   t5[480] := -0.013076;
   t5[481] := -0.0088184;
   t5[482] := -0.0046621;
   t5[483] := -0.0006165;
   t5[484] := 0.0033093;
   t5[485] := 0.0071061;
   t5[486] := 0.0107645;
   t5[487] := 0.0142754;
   t5[488] := 0.0176295;
   t5[489] := 0.0208177;
   t5[490] := 0.023831;
   t5[491] := 0.0266696;
   t5[492] := 0.0293428;
   t5[493] := 0.0318604;
   t5[494] := 0.0342322;
   t5[495] := -0.0208986;
   t5[496] := -0.0225395;
   t5[497] := -0.0240864;
   t5[498] := -0.0255261;
   t5[499] := -0.0268454;
   t5[500] := -0.0280312;
   t5[501] := -0.0290703;
   t5[502] := -0.0299495;
   t5[503] := -0.0306555;
   t5[504] := -0.0311752;
   t5[505] := -0.0314958;
   t5[506] := -0.0316138;
   t5[507] := -0.0315351;
   t5[508] := -0.0312663;
   t5[509] := -0.0308137;
   t5[510] := -0.0136591;
   t5[511] := -0.0122989;
   t5[512] := -0.0110547;
   t5[513] := -0.0099303;
   t5[514] := -0.0089297;
   t5[515] := -0.0080568;
   t5[516] := -0.0073155;
   t5[517] := -0.0067099;
   t5[518] := -0.0062437;
   t5[519] := -0.0059209;
   t5[520] := -0.0057453;
   t5[521] := -0.0057154;
   t5[522] := -0.0058246;
   t5[523] := -0.006066;
   t5[524] := -0.0064327;
   t5[525] := -0.014299;
   t5[526] := -0.0104196;
   t5[527] := -0.0064601;
   t5[528] := -0.0024202;
   t5[529] := 0.0017005;
   t5[530] := 0.0059023;
   t5[531] := 0.0101856;
   t5[532] := 0.0145506;
   t5[533] := 0.0189979;
   t5[534] := 0.0235277;
   t5[535] := 0.0281401;
   t5[536] := 0.0328307;
   t5[537] := 0.0375902;
   t5[538] := 0.042409;
   t5[539] := 0.0472775;
   t5[540] := -0.0809446;
   t5[541] := -0.0816613;
   t5[542] := -0.0823782;
   t5[543] := -0.0831006;
   t5[544] := -0.0838339;
   t5[545] := -0.0845833;
   t5[546] := -0.0853541;
   t5[547] := -0.0861518;
   t5[548] := -0.0869815;
   t5[549] := -0.0878487;
   t5[550] := -0.0887583;
   t5[551] := -0.0897094;
   t5[552] := -0.0906944;
   t5[553] := -0.0917059;
   t5[554] := -0.092736;
   t5[555] := 0.0001257;
   t5[556] := 0.0029497;
   t5[557] := 0.0057871;
   t5[558] := 0.0086392;
   t5[559] := 0.0115078;
   t5[560] := 0.0143943;
   t5[561] := 0.0173003;
   t5[562] := 0.0202273;
   t5[563] := 0.0231768;
   t5[564] := 0.0261505;
   t5[565] := 0.0291498;
   t5[566] := 0.0321767;
   t5[567] := 0.0352333;
   t5[568] := 0.0383218;
   t5[569] := 0.0414445;
   t5[570] := -0.0673197;
   t5[571] := -0.0670321;
   t5[572] := -0.0666434;
   t5[573] := -0.0661514;
   t5[574] := -0.0655542;
   t5[575] := -0.0648497;
   t5[576] := -0.0640358;
   t5[577] := -0.0631107;
   t5[578] := -0.0620721;
   t5[579] := -0.0609182;
   t5[580] := -0.0596471;
   t5[581] := -0.0582624;
   t5[582] := -0.0567733;
   t5[583] := -0.0551894;
   t5[584] := -0.05352;
   t5[585] := 0.0792828;
   t5[586] := 0.0762561;
   t5[587] := 0.073232;
   t5[588] := 0.0702186;
   t5[589] := 0.067224;
   t5[590] := 0.0642562;
   t5[591] := 0.0613231;
   t5[592] := 0.058433;
   t5[593] := 0.0555937;
   t5[594] := 0.0528132;
   t5[595] := 0.0500996;
   t5[596] := 0.0474569;
   t5[597] := 0.0448857;
   t5[598] := 0.042386;
   t5[599] := 0.0399582;
   t5[600] := -0.1993882;
   t5[601] := -0.1970195;
   t5[602] := -0.1945705;
   t5[603] := -0.1920432;
   t5[604] := -0.1894396;
   t5[605] := -0.1867614;
   t5[606] := -0.1840106;
   t5[607] := -0.1811892;
   t5[608] := -0.1782989;
   t5[609] := -0.1753418;
   t5[610] := -0.1723197;
   t5[611] := -0.1692367;
   t5[612] := -0.1660989;
   t5[613] := -0.1629122;
   t5[614] := -0.159683;
   t5[615] := -0.110986;
   t5[616] := -0.112907;
   t5[617] := -0.1145904;
   t5[618] := -0.11603;
   t5[619] := -0.1172196;
   t5[620] := -0.118153;
   t5[621] := -0.1188239;
   t5[622] := -0.119226;
   t5[623] := -0.1193531;
   t5[624] := -0.1191991;
   t5[625] := -0.1187581;
   t5[626] := -0.1180348;
   t5[627] := -0.1170453;
   t5[628] := -0.1158056;
   t5[629] := -0.1143322;
   t5[630] := -0.0163093;
   t5[631] := -0.0198292;
   t5[632] := -0.0232166;
   t5[633] := -0.0264609;
   t5[634] := -0.0295518;
   t5[635] := -0.0324788;
   t5[636] := -0.0352314;
   t5[637] := -0.0377992;
   t5[638] := -0.0401717;
   t5[639] := -0.0423386;
   t5[640] := -0.0442896;
   t5[641] := -0.0460239;
   t5[642] := -0.0475501;
   t5[643] := -0.0488771;
   t5[644] := -0.0500139;
   t5[645] := 0.0848828;
   t5[646] := 0.0819437;
   t5[647] := 0.0790844;
   t5[648] := 0.0763136;
   t5[649] := 0.0736399;
   t5[650] := 0.0710721;
   t5[651] := 0.0686188;
   t5[652] := 0.0662886;
   t5[653] := 0.0640904;
   t5[654] := 0.0620326;
   t5[655] := 0.0601237;
   t5[656] := 0.0583629;
   t5[657] := 0.05674;
   t5[658] := 0.0552444;
   t5[659] := 0.0538658;
   t5[660] := -0.0819279;
   t5[661] := -0.0837696;
   t5[662] := -0.085415;
   t5[663] := -0.0868444;
   t5[664] := -0.088038;
   t5[665] := -0.0889764;
   t5[666] := -0.0896396;
   t5[667] := -0.0900081;
   t5[668] := -0.0900622;
   t5[669] := -0.0897822;
   t5[670] := -0.0891493;
   t5[671] := -0.0881638;
   t5[672] := -0.0868462;
   t5[673] := -0.0852177;
   t5[674] := -0.0832996;
   t5[675] := -0.0222091;
   t5[676] := -0.019204;
   t5[677] := -0.0163363;
   t5[678] := -0.0136269;
   t5[679] := -0.0110964;
   t5[680] := -0.0087656;
   t5[681] := -0.0066552;
   t5[682] := -0.004786;
   t5[683] := -0.0031786;
   t5[684] := -0.0018538;
   t5[685] := -0.0008317;
   t5[686] := -0.0001178;
   t5[687] := 0.0002977;
   t5[688] := 0.0004254;
   t5[689] := 0.0002755;
   t5[690] := -0.0469918;
   t5[691] := -0.0436484;
   t5[692] := -0.0405246;
   t5[693] := -0.0376308;
   t5[694] := -0.0349775;
   t5[695] := -0.0325752;
   t5[696] := -0.0304344;
   t5[697] := -0.0285657;
   t5[698] := -0.0269795;
   t5[699] := -0.0256863;
   t5[700] := -0.0246962;
   t5[701] := -0.0240066;
   t5[702] := -0.0236022;
   t5[703] := -0.0234672;
   t5[704] := -0.0235855;
   t5[705] := 0.0315658;
   t5[706] := 0.0328791;
   t5[707] := 0.0340612;
   t5[708] := 0.0351116;
   t5[709] := 0.0360298;
   t5[710] := 0.0368152;
   t5[711] := 0.0374672;
   t5[712] := 0.0379854;
   t5[713] := 0.0383692;
   t5[714] := 0.038618;
   t5[715] := 0.0387315;
   t5[716] := 0.0387144;
   t5[717] := 0.0385764;
   t5[718] := 0.0383273;
   t5[719] := 0.0379772;
   t5[720] := 0.0589575;
   t5[721] := 0.0571638;
   t5[722] := 0.0552337;
   t5[723] := 0.0531697;
   t5[724] := 0.0509741;
   t5[725] := 0.0486495;
   t5[726] := 0.0461984;
   t5[727] := 0.0436231;
   t5[728] := 0.0409261;
   t5[729] := 0.03811;
   t5[730] := 0.0351772;
   t5[731] := 0.0321336;
   t5[732] := 0.0289883;
   t5[733] := 0.0257505;
   t5[734] := 0.0224294;
   t5[735] := -0.0370074;
   t5[736] := -0.0344528;
   t5[737] := -0.0317711;
   t5[738] := -0.0289586;
   t5[739] := -0.0260112;
   t5[740] := -0.022925;
   t5[741] := -0.0196963;
   t5[742] := -0.016321;
   t5[743] := -0.0127952;
   t5[744] := -0.0091151;
   t5[745] := -0.005277;
   t5[746] := -0.0012858;
   t5[747] := 0.0028455;
   t5[748] := 0.007103;
   t5[749] := 0.0114734;
   t5[750] := -0.0503424;
   t5[751] := -0.0554995;
   t5[752] := -0.0605443;
   t5[753] := -0.0654624;
   t5[754] := -0.0702395;
   t5[755] := -0.0748614;
   t5[756] := -0.0793139;
   t5[757] := -0.0835825;
   t5[758] := -0.087653;
   t5[759] := -0.0915111;
   t5[760] := -0.095143;
   t5[761] := -0.0985424;
   t5[762] := -0.1017114;
   t5[763] := -0.1046524;
   t5[764] := -0.1073677;
   t5[765] := -0.1648159;
   t5[766] := -0.1596806;
   t5[767] := -0.1543417;
   t5[768] := -0.1488126;
   t5[769] := -0.1431066;
   t5[770] := -0.1372371;
   t5[771] := -0.1312175;
   t5[772] := -0.1250611;
   t5[773] := -0.1187812;
   t5[774] := -0.1123913;
   t5[775] := -0.1059046;
   t5[776] := -0.0993333;
   t5[777] := -0.0926887;
   t5[778] := -0.0859816;
   t5[779] := -0.0792232;
   t5[780] := -0.0904827;
   t5[781] := -0.0898896;
   t5[782] := -0.0893127;
   t5[783] := -0.0887551;
   t5[784] := -0.0882202;
   t5[785] := -0.0877112;
   t5[786] := -0.0872314;
   t5[787] := -0.0867841;
   t5[788] := -0.0863725;
   t5[789] := -0.0859999;
   t5[790] := -0.0856695;
   t5[791] := -0.0853802;
   t5[792] := -0.0851272;
   t5[793] := -0.0849053;
   t5[794] := -0.0847093;
   t5[795] := -0.0673839;
   t5[796] := -0.0627446;
   t5[797] := -0.0580462;
   t5[798] := -0.0533;
   t5[799] := -0.0485171;
   t5[800] := -0.0437086;
   t5[801] := -0.0388857;
   t5[802] := -0.0340594;
   t5[803] := -0.0292411;
   t5[804] := -0.0244417;
   t5[805] := -0.0196723;
   t5[806] := -0.0149416;
   t5[807] := -0.0102555;
   t5[808] := -0.0056201;
   t5[809] := -0.0010412;
   t5[810] := 0.075334;
   t5[811] := 0.0749833;
   t5[812] := 0.0743661;
   t5[813] := 0.0734706;
   t5[814] := 0.072285;
   t5[815] := 0.0707974;
   t5[816] := 0.068996;
   t5[817] := 0.0668689;
   t5[818] := 0.0644045;
   t5[819] := 0.0615908;
   t5[820] := 0.0584166;
   t5[821] := 0.0548866;
   t5[822] := 0.0510212;
   t5[823] := 0.0468419;
   t5[824] := 0.04237;
   t5[825] := -0.1063465;
   t5[826] := -0.1045535;
   t5[827] := -0.1026798;
   t5[828] := -0.1007291;
   t5[829] := -0.0987055;
   t5[830] := -0.0966127;
   t5[831] := -0.0944546;
   t5[832] := -0.092235;
   t5[833] := -0.0899577;
   t5[834] := -0.0876267;
   t5[835] := -0.0852457;
   t5[836] := -0.0828167;
   t5[837] := -0.0803401;
   t5[838] := -0.077816;
   t5[839] := -0.0752449;
   t5[840] := 0.0025241;
   t5[841] := 0.0003729;
   t5[842] := -0.0018117;
   t5[843] := -0.0040243;
   t5[844] := -0.0062591;
   t5[845] := -0.0085107;
   t5[846] := -0.0107734;
   t5[847] := -0.0130416;
   t5[848] := -0.0153097;
   t5[849] := -0.0175722;
   t5[850] := -0.0198235;
   t5[851] := -0.0220606;
   t5[852] := -0.0242824;
   t5[853] := -0.0264882;
   t5[854] := -0.0286772;
   t5[855] := -0.0587365;
   t5[856] := -0.0658987;
   t5[857] := -0.0729648;
   t5[858] := -0.07991;
   t5[859] := -0.0867094;
   t5[860] := -0.0933378;
   t5[861] := -0.0997704;
   t5[862] := -0.1059823;
   t5[863] := -0.1119484;
   t5[864] := -0.1176438;
   t5[865] := -0.1230443;
   t5[866] := -0.1281403;
   t5[867] := -0.1329374;
   t5[868] := -0.137442;
   t5[869] := -0.1416606;
   t5[870] := -0.0241061;
   t5[871] := -0.0227329;
   t5[872] := -0.0212774;
   t5[873] := -0.0197337;
   t5[874] := -0.0180954;
   t5[875] := -0.0163565;
   t5[876] := -0.0145109;
   t5[877] := -0.0125525;
   t5[878] := -0.0104751;
   t5[879] := -0.0082726;
   t5[880] := -0.0059392;
   t5[881] := -0.0034767;
   t5[882] := -0.0008946;
   t5[883] := 0.001797;
   t5[884] := 0.0045883;
   t5[885] := -0.016338;
   t5[886] := -0.0135221;
   t5[887] := -0.0107115;
   t5[888] := -0.0079037;
   t5[889] := -0.0050963;
   t5[890] := -0.0022869;
   t5[891] := 0.0005271;
   t5[892] := 0.0033482;
   t5[893] := 0.0061787;
   t5[894] := 0.0090212;
   t5[895] := 0.011878;
   t5[896] := 0.0147486;
   t5[897] := 0.0176293;
   t5[898] := 0.0205164;
   t5[899] := 0.0234063;
   t5[900] := -0.0519279;
   t5[901] := -0.056473;
   t5[902] := -0.0609004;
   t5[903] := -0.0652012;
   t5[904] := -0.0693667;
   t5[905] := -0.0733882;
   t5[906] := -0.0772569;
   t5[907] := -0.0809641;
   t5[908] := -0.0845011;
   t5[909] := -0.087859;
   t5[910] := -0.0910294;
   t5[911] := -0.0940104;
   t5[912] := -0.0968068;
   t5[913] := -0.0994238;
   t5[914] := -0.1018665;
   t5[915] := 0.142846;
   t5[916] := 0.1405271;
   t5[917] := 0.1380653;
   t5[918] := 0.1354591;
   t5[919] := 0.1327065;
   t5[920] := 0.129806;
   t5[921] := 0.1267559;
   t5[922] := 0.1235543;
   t5[923] := 0.1201996;
   t5[924] := 0.11669;
   t5[925] := 0.1130242;
   t5[926] := 0.109206;
   t5[927] := 0.1052453;
   t5[928] := 0.1011521;
   t5[929] := 0.0969364;
   t5[930] := -0.0299947;
   t5[931] := -0.0294521;
   t5[932] := -0.0288785;
   t5[933] := -0.0282723;
   t5[934] := -0.0276319;
   t5[935] := -0.0269553;
   t5[936] := -0.0262411;
   t5[937] := -0.0254874;
   t5[938] := -0.0246926;
   t5[939] := -0.0238549;
   t5[940] := -0.0229728;
   t5[941] := -0.0220476;
   t5[942] := -0.0210837;
   t5[943] := -0.0200855;
   t5[944] := -0.0190576;
   t5[945] := -0.0100999;
   t5[946] := -0.0030712;
   t5[947] := 0.0037406;
   t5[948] := 0.0103103;
   t5[949] := 0.0166126;
   t5[950] := 0.0226221;
   t5[951] := 0.0283136;
   t5[952] := 0.0336617;
   t5[953] := 0.038641;
   t5[954] := 0.0432264;
   t5[955] := 0.0473932;
   t5[956] := 0.0511381;
   t5[957] := 0.054479;
   t5[958] := 0.0574348;
   t5[959] := 0.0600244;
   w6[0] := 0.0254122;
   w6[1] := -0.4251655;
   w6[2] := -0.4513899;
   w6[3] := 0.0262705;
   w6[4] := 0.3702881;
   w6[5] := -0.1208161;
   w6[6] := -0.2231239;
   w6[7] := 0.2512441;
   w6[8] := -0.3278799;
   w6[9] := 0.2889541;
   w6[10] := -0.0654242;
   w6[11] := 0.1067281;
   w6[12] := 0.2623815;
   w6[13] := -0.1798091;
   w6[14] := -0.3070911;
   w6[15] := -0.4204447;
   w6[16] := 0.5762351;
   w6[17] := -1.090657;
   w6[18] := -0.2690518;
   w6[19] := -0.6730261;
   w6[20] := -0.0514923;
   w6[21] := -0.4457789;
   w6[22] := 0.5072183;
   w6[23] := -0.0549661;
   w6[24] := 0.3812394;
   w6[25] := -0.606307;
   w6[26] := 0.1917919;
   w6[27] := 0.1525442;
   w6[28] := -0.4219312;
   w6[29] := 0.338313;
   w6[30] := 0.1919874;
   w6[31] := -0.3457294;
   w6[32] := 0.1728978;
   w6[33] := 0.5825878;
   w6[34] := 0.7331663;
   w6[35] := 0.4268312;
   w6[36] := -0.0077422;
   w6[37] := 0.4766487;
   w6[38] := 0.102607;
   w6[39] := -0.5723706;
   w6[40] := 0.0728498;
   w6[41] := 0.4253429;
   w6[42] := -0.3637053;
   w6[43] := -0.6206156;
   w6[44] := 0.2656944;
   w6[45] := -0.3130539;
   w6[46] := 0.2033212;
   w6[47] := 0.1327122;
   w6[48] := -0.709101;
   w6[49] := 0.7231103;
   w6[50] := -0.2214241;
   w6[51] := 0.4491622;
   w6[52] := -0.3655713;
   w6[53] := 0.4263724;
   w6[54] := 0.0266531;
   w6[55] := 0.4637966;
   w6[56] := -0.3418979;
   w6[57] := -0.2391363;
   w6[58] := 0.4152579;
   w6[59] := 0.2146362;
   w6[60] := -0.3901598;
   w6[61] := -0.1938754;
   w6[62] := -0.561949;
   w6[63] := 0.4047181;
END_DATA_BLOCK

DATA_BLOCK "NeuroPLC_MLP_Weights"   // DB3
{ S7_Optimized_Access := 'FALSE' }
VERSION : 0.1
   VAR
      w0 : Array[0..895] of Real;   // W(32x28)
      b1 : Array[0..31] of Real;   // bias(32)
      w2 : Array[0..511] of Real;   // W(16x32)
      b3 : Array[0..15] of Real;   // bias(16)
      w4 : Array[0..63] of Real;   // W(4x16)
      b5 : Array[0..3] of Real;   // bias(4)
   END_VAR
BEGIN
   w0[0] := 0.5694862;
   w0[1] := -0.0095692;
   w0[2] := 0.7619486;
   w0[3] := 0.2215109;
   w0[4] := -0.3561512;
   w0[5] := -0.2522623;
   w0[6] := 0.2582799;
   w0[7] := 0.0099258;
   w0[8] := 0.3836571;
   w0[9] := -0.0658457;
   w0[10] := 0.1010401;
   w0[11] := -0.2984352;
   w0[12] := 0.1934527;
   w0[13] := -0.264014;
   w0[14] := 0.1362384;
   w0[15] := -0.0190728;
   w0[16] := -0.2375232;
   w0[17] := -0.1084833;
   w0[18] := -0.3846658;
   w0[19] := 0.3771667;
   w0[20] := -0.1136759;
   w0[21] := -0.1259104;
   w0[22] := -0.1682155;
   w0[23] := 0.4097499;
   w0[24] := -0.2194012;
   w0[25] := -0.2356472;
   w0[26] := -0.1771912;
   w0[27] := 0.1675407;
   w0[28] := 0.1454716;
   w0[29] := -0.3696787;
   w0[30] := -0.2783369;
   w0[31] := -0.1873165;
   w0[32] := 0.0781848;
   w0[33] := -0.3527579;
   w0[34] := -0.2131715;
   w0[35] := -0.413968;
   w0[36] := -0.5927966;
   w0[37] := 0.3198802;
   w0[38] := -0.5640871;
   w0[39] := -0.2003005;
   w0[40] := 0.1832723;
   w0[41] := 0.2237836;
   w0[42] := 0.1929916;
   w0[43] := 0.2185234;
   w0[44] := 0.1214973;
   w0[45] := 0.0208249;
   w0[46] := 0.2776418;
   w0[47] := 0.6831574;
   w0[48] := -0.1655439;
   w0[49] := -0.2658227;
   w0[50] := -0.2709237;
   w0[51] := 0.098671;
   w0[52] := 0.1128972;
   w0[53] := -0.2047481;
   w0[54] := -0.3872808;
   w0[55] := 0.1596099;
   w0[56] := -0.2523361;
   w0[57] := 0.2758174;
   w0[58] := 0.2686562;
   w0[59] := -0.5177624;
   w0[60] := -0.1129441;
   w0[61] := -0.21921;
   w0[62] := 0.3343761;
   w0[63] := -0.0422801;
   w0[64] := -0.3068857;
   w0[65] := 0.2210509;
   w0[66] := -0.5496964;
   w0[67] := 0.3709493;
   w0[68] := 0.0747587;
   w0[69] := -0.1170707;
   w0[70] := -0.319511;
   w0[71] := 0.0277475;
   w0[72] := -0.2577946;
   w0[73] := 0.0641775;
   w0[74] := 0.2055912;
   w0[75] := 0.6039576;
   w0[76] := -0.5010191;
   w0[77] := 0.0377836;
   w0[78] := 0.2038942;
   w0[79] := -0.0376425;
   w0[80] := 0.1546009;
   w0[81] := 0.3260912;
   w0[82] := -0.1506072;
   w0[83] := 0.0569262;
   w0[84] := -0.1928782;
   w0[85] := -0.198454;
   w0[86] := -0.0539345;
   w0[87] := 0.3094364;
   w0[88] := 0.2289592;
   w0[89] := -0.425005;
   w0[90] := -0.0399776;
   w0[91] := 0.0658291;
   w0[92] := 0.2534966;
   w0[93] := -0.0973715;
   w0[94] := -0.3647969;
   w0[95] := -0.015606;
   w0[96] := -0.5209337;
   w0[97] := 0.2564455;
   w0[98] := 0.1338747;
   w0[99] := 0.3502659;
   w0[100] := -0.3756513;
   w0[101] := 0.253089;
   w0[102] := 0.0984663;
   w0[103] := 0.6602526;
   w0[104] := 0.3365156;
   w0[105] := -0.2521311;
   w0[106] := 0.0946512;
   w0[107] := -0.6085349;
   w0[108] := -0.5372492;
   w0[109] := 0.0455726;
   w0[110] := -0.0786947;
   w0[111] := 0.0370381;
   w0[112] := -0.585835;
   w0[113] := -0.7779619;
   w0[114] := -0.7385424;
   w0[115] := -0.207106;
   w0[116] := 0.2831336;
   w0[117] := 0.3243212;
   w0[118] := 0.2366221;
   w0[119] := -0.2105746;
   w0[120] := -0.3834608;
   w0[121] := -0.6828474;
   w0[122] := 0.1007835;
   w0[123] := 0.0381121;
   w0[124] := 0.3126857;
   w0[125] := 0.0975034;
   w0[126] := 0.0499541;
   w0[127] := -0.0530838;
   w0[128] := 0.0799674;
   w0[129] := -0.1505451;
   w0[130] := -0.4892448;
   w0[131] := -0.3954702;
   w0[132] := 0.1594549;
   w0[133] := 0.2307071;
   w0[134] := -0.0041823;
   w0[135] := 0.5944483;
   w0[136] := -0.2759206;
   w0[137] := -0.4257804;
   w0[138] := -0.3279784;
   w0[139] := -0.297798;
   w0[140] := 0.0038754;
   w0[141] := 0.3761657;
   w0[142] := 0.4177073;
   w0[143] := 0.0741864;
   w0[144] := 0.3750937;
   w0[145] := 0.2039272;
   w0[146] := -0.2429399;
   w0[147] := -0.3849822;
   w0[148] := 0.1600508;
   w0[149] := -0.1581226;
   w0[150] := -0.0233814;
   w0[151] := -0.1151747;
   w0[152] := -0.5731639;
   w0[153] := -0.0274457;
   w0[154] := 0.1195597;
   w0[155] := -0.2395748;
   w0[156] := 0.2293357;
   w0[157] := -0.0251415;
   w0[158] := 0.3937997;
   w0[159] := -0.1454628;
   w0[160] := -0.0673693;
   w0[161] := 0.2948158;
   w0[162] := 0.5630679;
   w0[163] := -0.3092144;
   w0[164] := 0.1832785;
   w0[165] := 0.004312;
   w0[166] := 0.0011036;
   w0[167] := 0.2549984;
   w0[168] := 0.1242365;
   w0[169] := -0.1573328;
   w0[170] := 0.1472307;
   w0[171] := 0.2971004;
   w0[172] := 0.1052006;
   w0[173] := 0.3616425;
   w0[174] := -0.1347494;
   w0[175] := -0.3794992;
   w0[176] := 0.5467421;
   w0[177] := -0.1476457;
   w0[178] := 0.3496484;
   w0[179] := -0.0583753;
   w0[180] := 0.2853532;
   w0[181] := -0.3058073;
   w0[182] := -0.1615329;
   w0[183] := -0.522915;
   w0[184] := 0.2140338;
   w0[185] := -0.2294949;
   w0[186] := 0.2921923;
   w0[187] := 0.0373898;
   w0[188] := 0.3493846;
   w0[189] := 0.5938788;
   w0[190] := 0.0955027;
   w0[191] := -0.1719695;
   w0[192] := 0.6582399;
   w0[193] := -0.491165;
   w0[194] := 0.126987;
   w0[195] := -0.412937;
   w0[196] := -0.273549;
   w0[197] := -0.215566;
   w0[198] := 0.4269275;
   w0[199] := -0.1273027;
   w0[200] := -0.2414422;
   w0[201] := -0.3611139;
   w0[202] := 0.6480063;
   w0[203] := 0.3808921;
   w0[204] := -0.2189153;
   w0[205] := 0.0094489;
   w0[206] := 0.6784652;
   w0[207] := 0.3757944;
   w0[208] := 0.5965886;
   w0[209] := 0.3704935;
   w0[210] := 0.3205929;
   w0[211] := 0.2190031;
   w0[212] := -0.3913886;
   w0[213] := 0.2046225;
   w0[214] := 0.7660633;
   w0[215] := 0.5648795;
   w0[216] := 0.0447379;
   w0[217] := -0.1363681;
   w0[218] := -0.1653181;
   w0[219] := -0.3211187;
   w0[220] := 0.0557173;
   w0[221] := -0.677563;
   w0[222] := 0.2077208;
   w0[223] := 0.1863764;
   w0[224] := 0.0122372;
   w0[225] := -0.1510706;
   w0[226] := -0.0393031;
   w0[227] := -0.237385;
   w0[228] := 0.3297745;
   w0[229] := -0.3327326;
   w0[230] := -0.1183226;
   w0[231] := 0.3871697;
   w0[232] := -0.448105;
   w0[233] := -0.2065133;
   w0[234] := 0.1012533;
   w0[235] := -0.2578072;
   w0[236] := 0.0634624;
   w0[237] := -0.1246978;
   w0[238] := 0.1465549;
   w0[239] := -0.5023389;
   w0[240] := 0.0640146;
   w0[241] := 0.1963426;
   w0[242] := 0.6648222;
   w0[243] := -0.6102669;
   w0[244] := -0.28719;
   w0[245] := -0.3684005;
   w0[246] := -0.4533643;
   w0[247] := -0.1819637;
   w0[248] := -0.3802012;
   w0[249] := 0.4682154;
   w0[250] := 0.1991423;
   w0[251] := 0.5698866;
   w0[252] := 0.3063245;
   w0[253] := 0.1672625;
   w0[254] := 0.261124;
   w0[255] := -0.6845852;
   w0[256] := -0.1005014;
   w0[257] := -0.6641653;
   w0[258] := -0.254451;
   w0[259] := 0.1954752;
   w0[260] := -0.2994281;
   w0[261] := 0.3571715;
   w0[262] := -0.0372742;
   w0[263] := -0.0310561;
   w0[264] := 0.1959654;
   w0[265] := -0.1060541;
   w0[266] := 0.3827632;
   w0[267] := -0.3923316;
   w0[268] := -0.592409;
   w0[269] := 0.0670658;
   w0[270] := 0.3532278;
   w0[271] := 0.6439264;
   w0[272] := 0.1193878;
   w0[273] := -0.5490641;
   w0[274] := -0.6517076;
   w0[275] := 0.2266813;
   w0[276] := 0.273508;
   w0[277] := 0.2562127;
   w0[278] := 0.3711089;
   w0[279] := -0.0201157;
   w0[280] := 0.5907255;
   w0[281] := 0.3026478;
   w0[282] := 0.087949;
   w0[283] := -0.1103418;
   w0[284] := 0.0830003;
   w0[285] := 0.0901832;
   w0[286] := 0.4872787;
   w0[287] := -0.4248994;
   w0[288] := 0.6916616;
   w0[289] := 0.0068263;
   w0[290] := 0.0377772;
   w0[291] := -0.345046;
   w0[292] := 0.5848706;
   w0[293] := -0.0756037;
   w0[294] := 0.0390328;
   w0[295] := -0.4139087;
   w0[296] := -0.1527735;
   w0[297] := -0.2285863;
   w0[298] := 0.3310088;
   w0[299] := 0.2031009;
   w0[300] := -0.5309294;
   w0[301] := -0.4607368;
   w0[302] := 0.1824918;
   w0[303] := -0.1911459;
   w0[304] := -0.1732452;
   w0[305] := -0.3283744;
   w0[306] := -0.0425148;
   w0[307] := -0.075475;
   w0[308] := -0.075183;
   w0[309] := -0.0057766;
   w0[310] := -0.0669558;
   w0[311] := -0.0518108;
   w0[312] := -0.1100485;
   w0[313] := 0.4202482;
   w0[314] := 0.1722786;
   w0[315] := 0.254064;
   w0[316] := -0.2125306;
   w0[317] := -0.3108644;
   w0[318] := -0.1653187;
   w0[319] := 0.0082027;
   w0[320] := 0.1613134;
   w0[321] := 0.5696448;
   w0[322] := 0.4734836;
   w0[323] := -0.1820288;
   w0[324] := -0.0202256;
   w0[325] := 0.2319008;
   w0[326] := 0.6178575;
   w0[327] := -0.1729726;
   w0[328] := -0.5705087;
   w0[329] := -0.4175466;
   w0[330] := -0.0846097;
   w0[331] := -0.4305633;
   w0[332] := -0.0297265;
   w0[333] := -0.2146564;
   w0[334] := -0.0228577;
   w0[335] := 0.4386194;
   w0[336] := 0.1366172;
   w0[337] := 0.1275948;
   w0[338] := 0.2872518;
   w0[339] := -0.046949;
   w0[340] := -0.3430789;
   w0[341] := -0.2333279;
   w0[342] := -0.0942715;
   w0[343] := -0.6695372;
   w0[344] := 0.3036573;
   w0[345] := 0.6706407;
   w0[346] := 0.4867018;
   w0[347] := 0.2229243;
   w0[348] := 0.1479198;
   w0[349] := 0.4786703;
   w0[350] := -0.1235309;
   w0[351] := -0.1444162;
   w0[352] := -0.1594525;
   w0[353] := 0.0118241;
   w0[354] := 0.3302614;
   w0[355] := 0.4612524;
   w0[356] := -0.1728074;
   w0[357] := -0.4940682;
   w0[358] := 0.266313;
   w0[359] := 0.4213447;
   w0[360] := 0.155972;
   w0[361] := 0.0927116;
   w0[362] := 0.2581408;
   w0[363] := 0.1484697;
   w0[364] := 0.5596921;
   w0[365] := 0.6450443;
   w0[366] := 0.2316463;
   w0[367] := -0.3064318;
   w0[368] := 0.315403;
   w0[369] := 0.2504337;
   w0[370] := 0.2270162;
   w0[371] := -0.2362736;
   w0[372] := -0.1822204;
   w0[373] := 0.7585521;
   w0[374] := 0.2454521;
   w0[375] := -0.3572387;
   w0[376] := 0.1800293;
   w0[377] := 0.1965537;
   w0[378] := 0.1946464;
   w0[379] := 0.1738928;
   w0[380] := -0.1159788;
   w0[381] := -0.1791228;
   w0[382] := 0.3109314;
   w0[383] := 0.1039406;
   w0[384] := -0.255849;
   w0[385] := -0.4132357;
   w0[386] := -0.1826324;
   w0[387] := -0.0949509;
   w0[388] := 0.075463;
   w0[389] := -0.4951166;
   w0[390] := -0.0366096;
   w0[391] := -0.5241205;
   w0[392] := 0.0701182;
   w0[393] := 0.5458165;
   w0[394] := -0.3082272;
   w0[395] := -0.162029;
   w0[396] := 0.2685293;
   w0[397] := -0.1115321;
   w0[398] := 0.5528188;
   w0[399] := 0.1818966;
   w0[400] := -0.270587;
   w0[401] := -0.4477837;
   w0[402] := -0.3260813;
   w0[403] := -0.1751753;
   w0[404] := 0.3439055;
   w0[405] := 0.369066;
   w0[406] := -0.0775537;
   w0[407] := -0.3291571;
   w0[408] := 0.396657;
   w0[409] := 0.3747428;
   w0[410] := 0.2037812;
   w0[411] := 0.506327;
   w0[412] := -0.0363616;
   w0[413] := -0.0945516;
   w0[414] := -0.2667596;
   w0[415] := -0.1880456;
   w0[416] := 0.2148547;
   w0[417] := -0.659289;
   w0[418] := -0.2238534;
   w0[419] := -0.2862469;
   w0[420] := -0.8308039;
   w0[421] := -0.4430834;
   w0[422] := -0.0302747;
   w0[423] := 0.091846;
   w0[424] := -0.3334551;
   w0[425] := -0.1804388;
   w0[426] := -0.1097601;
   w0[427] := 0.3427432;
   w0[428] := 0.0736062;
   w0[429] := -0.6790179;
   w0[430] := -0.243052;
   w0[431] := -0.2084594;
   w0[432] := 0.1491454;
   w0[433] := -0.0083196;
   w0[434] := 0.2553293;
   w0[435] := 0.1678275;
   w0[436] := 0.0936099;
   w0[437] := 0.1736043;
   w0[438] := -0.5376837;
   w0[439] := -0.4510113;
   w0[440] := -0.3174161;
   w0[441] := 0.2371299;
   w0[442] := 0.3883051;
   w0[443] := 0.3464468;
   w0[444] := 0.1098732;
   w0[445] := 0.0205052;
   w0[446] := -0.2641115;
   w0[447] := -0.3012585;
   w0[448] := -0.5463231;
   w0[449] := -0.0684724;
   w0[450] := -0.1422806;
   w0[451] := -0.2644515;
   w0[452] := -0.4767578;
   w0[453] := -0.4182616;
   w0[454] := -0.4673964;
   w0[455] := -0.0129319;
   w0[456] := -0.5374129;
   w0[457] := -0.1050398;
   w0[458] := 0.0632549;
   w0[459] := 0.0568505;
   w0[460] := 0.2111508;
   w0[461] := 0.3917949;
   w0[462] := -0.0330271;
   w0[463] := 0.2814879;
   w0[464] := -0.3214771;
   w0[465] := 0.343051;
   w0[466] := -0.3870021;
   w0[467] := -0.4042188;
   w0[468] := 0.1747253;
   w0[469] := 0.3262924;
   w0[470] := 0.5594077;
   w0[471] := 0.0277393;
   w0[472] := -0.2604083;
   w0[473] := 0.0503597;
   w0[474] := 0.3725081;
   w0[475] := -0.0544451;
   w0[476] := 0.0951887;
   w0[477] := -0.5271522;
   w0[478] := -0.3720489;
   w0[479] := 0.0333015;
   w0[480] := 0.3407656;
   w0[481] := -0.0524092;
   w0[482] := -0.394772;
   w0[483] := 0.0632993;
   w0[484] := -0.4918242;
   w0[485] := -0.0408889;
   w0[486] := 0.5603451;
   w0[487] := 0.3429145;
   w0[488] := -0.0672607;
   w0[489] := -0.3218429;
   w0[490] := -0.3621323;
   w0[491] := -0.5524946;
   w0[492] := 0.3105496;
   w0[493] := 0.3352183;
   w0[494] := -0.6259544;
   w0[495] := -0.1107638;
   w0[496] := 0.0901521;
   w0[497] := 0.00385;
   w0[498] := 0.5420415;
   w0[499] := 0.2380718;
   w0[500] := -0.0511688;
   w0[501] := -0.077146;
   w0[502] := -0.0791493;
   w0[503] := -0.1069665;
   w0[504] := 0.6399192;
   w0[505] := -0.0014034;
   w0[506] := 0.3290343;
   w0[507] := -0.3565734;
   w0[508] := 0.2305476;
   w0[509] := -0.0417552;
   w0[510] := 0.294279;
   w0[511] := -0.1355964;
   w0[512] := 0.0557771;
   w0[513] := 0.3271682;
   w0[514] := -0.3025698;
   w0[515] := 0.28975;
   w0[516] := 0.1278277;
   w0[517] := -0.1560617;
   w0[518] := 0.2582703;
   w0[519] := -0.0549245;
   w0[520] := -0.0921321;
   w0[521] := 0.4996554;
   w0[522] := 0.0836308;
   w0[523] := 0.2032579;
   w0[524] := -0.1741465;
   w0[525] := -0.2436171;
   w0[526] := -0.3661414;
   w0[527] := -0.2924559;
   w0[528] := -0.4407195;
   w0[529] := 0.2304931;
   w0[530] := -0.2509898;
   w0[531] := -0.688146;
   w0[532] := 0.1500384;
   w0[533] := 0.4429501;
   w0[534] := 0.5444623;
   w0[535] := 0.0644146;
   w0[536] := 0.1564979;
   w0[537] := 0.1936211;
   w0[538] := -0.2217757;
   w0[539] := 0.163296;
   w0[540] := 0.0949209;
   w0[541] := 0.5449093;
   w0[542] := 0.3260632;
   w0[543] := 0.4177442;
   w0[544] := -0.1678705;
   w0[545] := -0.4614883;
   w0[546] := -0.1780888;
   w0[547] := 0.0282706;
   w0[548] := -0.3548764;
   w0[549] := 0.1119965;
   w0[550] := -0.6278588;
   w0[551] := -0.2857478;
   w0[552] := 0.3291071;
   w0[553] := -0.2958602;
   w0[554] := -0.2171935;
   w0[555] := 0.0488607;
   w0[556] := -0.2721503;
   w0[557] := -0.0109805;
   w0[558] := -0.2872001;
   w0[559] := -0.3800366;
   w0[560] := 0.7377275;
   w0[561] := 0.5175216;
   w0[562] := 0.4534726;
   w0[563] := 0.2131705;
   w0[564] := 0.1694544;
   w0[565] := 0.1088488;
   w0[566] := 0.2956495;
   w0[567] := -0.1219863;
   w0[568] := 0.4281839;
   w0[569] := 0.0482728;
   w0[570] := 0.326145;
   w0[571] := 0.0147065;
   w0[572] := 0.0197347;
   w0[573] := -0.2837075;
   w0[574] := -0.2223815;
   w0[575] := -0.3011971;
   w0[576] := 0.4010099;
   w0[577] := 0.3606303;
   w0[578] := 0.5675586;
   w0[579] := -0.1933776;
   w0[580] := 0.1411208;
   w0[581] := 0.4412328;
   w0[582] := -0.3157989;
   w0[583] := 0.0737199;
   w0[584] := 0.2547267;
   w0[585] := -0.4104514;
   w0[586] := 0.3333948;
   w0[587] := 0.0244799;
   w0[588] := 0.3485871;
   w0[589] := -0.1856655;
   w0[590] := -0.2338329;
   w0[591] := -0.2214157;
   w0[592] := 0.4647014;
   w0[593] := -0.3053385;
   w0[594] := -0.1758788;
   w0[595] := -0.2062785;
   w0[596] := 0.4421045;
   w0[597] := 0.290327;
   w0[598] := 0.2819436;
   w0[599] := -0.3433319;
   w0[600] := -0.0214767;
   w0[601] := 0.5416198;
   w0[602] := -0.014361;
   w0[603] := -0.1832658;
   w0[604] := -0.5633022;
   w0[605] := -0.1308155;
   w0[606] := 0.1253684;
   w0[607] := -0.346004;
   w0[608] := -0.0773746;
   w0[609] := -0.0179889;
   w0[610] := -0.3036036;
   w0[611] := 0.0990553;
   w0[612] := -0.2073587;
   w0[613] := 0.0275394;
   w0[614] := 0.0471204;
   w0[615] := -0.0187443;
   w0[616] := 0.4038751;
   w0[617] := 0.0922068;
   w0[618] := -0.2135524;
   w0[619] := -0.4082574;
   w0[620] := -0.035856;
   w0[621] := -0.1610684;
   w0[622] := -0.4163499;
   w0[623] := 0.246724;
   w0[624] := 0.0747931;
   w0[625] := 0.3987921;
   w0[626] := 0.1632655;
   w0[627] := -0.3848493;
   w0[628] := 0.1649167;
   w0[629] := -0.6442378;
   w0[630] := -0.4510081;
   w0[631] := -0.2822698;
   w0[632] := 0.4664556;
   w0[633] := -0.2991767;
   w0[634] := -0.0362801;
   w0[635] := -0.3327457;
   w0[636] := -0.3074295;
   w0[637] := 0.1606831;
   w0[638] := -0.0541677;
   w0[639] := -0.5748461;
   w0[640] := 0.3949239;
   w0[641] := -0.2336025;
   w0[642] := -0.0525538;
   w0[643] := 0.3131756;
   w0[644] := -0.0032524;
   w0[645] := -0.0003879;
   w0[646] := 0.3644529;
   w0[647] := 0.3278647;
   w0[648] := -0.0496909;
   w0[649] := -0.0200011;
   w0[650] := 0.4739185;
   w0[651] := -0.388666;
   w0[652] := 0.085598;
   w0[653] := -0.4665208;
   w0[654] := 0.4008028;
   w0[655] := -0.54488;
   w0[656] := -0.4093939;
   w0[657] := -0.132936;
   w0[658] := 0.2988919;
   w0[659] := -0.0788539;
   w0[660] := 0.028211;
   w0[661] := -0.1015701;
   w0[662] := 0.5736219;
   w0[663] := -0.2615215;
   w0[664] := 0.0237927;
   w0[665] := 0.0321014;
   w0[666] := -0.1239056;
   w0[667] := -0.2004481;
   w0[668] := -0.0194097;
   w0[669] := -0.1323835;
   w0[670] := -0.0777957;
   w0[671] := 0.0366594;
   w0[672] := 0.1079154;
   w0[673] := 0.4157223;
   w0[674] := -0.2902254;
   w0[675] := 0.4283061;
   w0[676] := 0.06503;
   w0[677] := 0.1249261;
   w0[678] := -0.2917063;
   w0[679] := -0.1270394;
   w0[680] := 0.0782463;
   w0[681] := 0.5982807;
   w0[682] := 0.101776;
   w0[683] := 0.1843081;
   w0[684] := -0.6125457;
   w0[685] := 0.2722199;
   w0[686] := -0.0728571;
   w0[687] := -0.5004624;
   w0[688] := 0.4432183;
   w0[689] := 0.491213;
   w0[690] := 0.0002442;
   w0[691] := -0.0942999;
   w0[692] := 0.5940161;
   w0[693] := -0.1235101;
   w0[694] := 0.3478113;
   w0[695] := 0.0345737;
   w0[696] := -0.0406947;
   w0[697] := 0.61514;
   w0[698] := 0.2030335;
   w0[699] := -0.323678;
   w0[700] := -0.6019017;
   w0[701] := -0.477923;
   w0[702] := -0.8101817;
   w0[703] := -0.2094196;
   w0[704] := -0.3149875;
   w0[705] := 0.3055148;
   w0[706] := -0.281898;
   w0[707] := 0.2800311;
   w0[708] := -0.8234739;
   w0[709] := -0.6584272;
   w0[710] := 0.2585062;
   w0[711] := 0.0584044;
   w0[712] := -0.5591815;
   w0[713] := -0.0547792;
   w0[714] := 0.0355113;
   w0[715] := 0.2701355;
   w0[716] := -0.5936313;
   w0[717] := 0.3193162;
   w0[718] := 0.1195579;
   w0[719] := 0.0537417;
   w0[720] := 0.6140408;
   w0[721] := 0.5008627;
   w0[722] := -0.0104372;
   w0[723] := 0.2329175;
   w0[724] := -0.0168664;
   w0[725] := 0.0332739;
   w0[726] := 0.3730388;
   w0[727] := 0.1635417;
   w0[728] := 0.7335413;
   w0[729] := 0.5691491;
   w0[730] := 0.0170918;
   w0[731] := 0.2825087;
   w0[732] := 0.0198349;
   w0[733] := 0.4498756;
   w0[734] := 0.410012;
   w0[735] := -0.2479021;
   w0[736] := 0.2850291;
   w0[737] := -0.1702987;
   w0[738] := -0.4980538;
   w0[739] := -0.0941117;
   w0[740] := 0.4272463;
   w0[741] := -0.2824812;
   w0[742] := 0.6535753;
   w0[743] := 0.2375765;
   w0[744] := 0.4509313;
   w0[745] := -0.0013205;
   w0[746] := 0.112706;
   w0[747] := -0.1239916;
   w0[748] := 0.3028973;
   w0[749] := 0.0927592;
   w0[750] := -0.3168923;
   w0[751] := 0.1611173;
   w0[752] := 0.4917028;
   w0[753] := 0.0417323;
   w0[754] := 0.3917417;
   w0[755] := -0.0557213;
   w0[756] := -0.2345485;
   w0[757] := 0.3833969;
   w0[758] := 0.3747815;
   w0[759] := -0.1519468;
   w0[760] := -0.3892233;
   w0[761] := -0.0699942;
   w0[762] := -0.3351573;
   w0[763] := -0.3026012;
   w0[764] := -0.1781991;
   w0[765] := 0.4689204;
   w0[766] := -0.1804391;
   w0[767] := -0.2284776;
   w0[768] := -0.3932275;
   w0[769] := 0.2445571;
   w0[770] := -0.1087966;
   w0[771] := -0.2825441;
   w0[772] := -0.230165;
   w0[773] := 0.5091258;
   w0[774] := -0.7006359;
   w0[775] := 0.0339814;
   w0[776] := 0.1417895;
   w0[777] := 0.1839303;
   w0[778] := 0.2910166;
   w0[779] := 0.1044962;
   w0[780] := 0.0580844;
   w0[781] := 0.615828;
   w0[782] := -0.0284938;
   w0[783] := 0.0542879;
   w0[784] := 0.1680317;
   w0[785] := 0.2264472;
   w0[786] := -0.2030084;
   w0[787] := 0.0756811;
   w0[788] := -0.2188872;
   w0[789] := -0.2264328;
   w0[790] := -0.1813061;
   w0[791] := -0.2645762;
   w0[792] := 0.4621922;
   w0[793] := -0.4514092;
   w0[794] := 0.3058094;
   w0[795] := 0.3434274;
   w0[796] := 0.3808913;
   w0[797] := -0.3231871;
   w0[798] := 0.2469297;
   w0[799] := -0.1890893;
   w0[800] := 0.0499585;
   w0[801] := -0.3218643;
   w0[802] := 0.6025205;
   w0[803] := 0.0650566;
   w0[804] := -0.2298092;
   w0[805] := 0.5071256;
   w0[806] := -0.2657916;
   w0[807] := -0.1830709;
   w0[808] := 0.041564;
   w0[809] := -0.1594847;
   w0[810] := -0.032166;
   w0[811] := -0.0346579;
   w0[812] := -0.381939;
   w0[813] := 0.2074234;
   w0[814] := 0.3919429;
   w0[815] := 0.0324158;
   w0[816] := -0.0215873;
   w0[817] := -0.132927;
   w0[818] := 0.0735578;
   w0[819] := 0.3148956;
   w0[820] := -0.443545;
   w0[821] := -0.3320747;
   w0[822] := -0.1767979;
   w0[823] := -0.4104172;
   w0[824] := 0.3253109;
   w0[825] := -0.1773608;
   w0[826] := -0.4930988;
   w0[827] := 0.3281353;
   w0[828] := 0.3916833;
   w0[829] := -0.1541856;
   w0[830] := 0.1263307;
   w0[831] := 0.0426248;
   w0[832] := -0.5533415;
   w0[833] := 0.0726361;
   w0[834] := -0.4881184;
   w0[835] := -0.1073755;
   w0[836] := -0.5946367;
   w0[837] := -0.574247;
   w0[838] := 0.1233901;
   w0[839] := -0.0872265;
   w0[840] := 0.2010813;
   w0[841] := 0.4012275;
   w0[842] := 0.3290967;
   w0[843] := 0.3005436;
   w0[844] := -0.0111396;
   w0[845] := -0.4794478;
   w0[846] := -0.0532993;
   w0[847] := -0.1733176;
   w0[848] := -0.1260332;
   w0[849] := 0.1089438;
   w0[850] := 0.0391418;
   w0[851] := -0.2468968;
   w0[852] := 0.4689822;
   w0[853] := -0.4640872;
   w0[854] := 0.2532913;
   w0[855] := -0.2343228;
   w0[856] := 0.2661497;
   w0[857] := -0.4386278;
   w0[858] := 0.0468966;
   w0[859] := -0.3265733;
   w0[860] := -0.1916417;
   w0[861] := 0.5178355;
   w0[862] := 0.2822486;
   w0[863] := -0.107772;
   w0[864] := 0.32863;
   w0[865] := -0.002981;
   w0[866] := -0.3535745;
   w0[867] := -0.1011055;
   w0[868] := 0.1318278;
   w0[869] := 0.0674391;
   w0[870] := 0.0591611;
   w0[871] := -0.1122496;
   w0[872] := 0.4686061;
   w0[873] := -0.4002847;
   w0[874] := 0.0749937;
   w0[875] := -0.1933431;
   w0[876] := 0.2702274;
   w0[877] := -0.1278288;
   w0[878] := -0.1761822;
   w0[879] := -0.2737747;
   w0[880] := 0.4466998;
   w0[881] := 0.0271071;
   w0[882] := 0.1916832;
   w0[883] := 0.4834492;
   w0[884] := 0.0259246;
   w0[885] := -0.489219;
   w0[886] := 0.2059345;
   w0[887] := -0.082233;
   w0[888] := -0.4142632;
   w0[889] := 0.54042;
   w0[890] := -0.1093403;
   w0[891] := 0.0186543;
   w0[892] := 0.6250578;
   w0[893] := -0.2241697;
   w0[894] := 0.308892;
   w0[895] := 0.1112378;
   b1[0] := -0.1609981;
   b1[1] := -0.0371174;
   b1[2] := 0.0221225;
   b1[3] := 0.0337845;
   b1[4] := 0.2616802;
   b1[5] := 0.1264098;
   b1[6] := 0.1833381;
   b1[7] := 0.1271529;
   b1[8] := 0.0488858;
   b1[9] := 0.0241906;
   b1[10] := -0.3121075;
   b1[11] := 0.0973287;
   b1[12] := -0.0882614;
   b1[13] := -0.3344531;
   b1[14] := -0.1306882;
   b1[15] := 0.151865;
   b1[16] := 0.0104939;
   b1[17] := -0.0685202;
   b1[18] := -0.095305;
   b1[19] := 0.0008646;
   b1[20] := 0.2513834;
   b1[21] := 0.0002911;
   b1[22] := 0.1923783;
   b1[23] := 0.1726166;
   b1[24] := 0.3154603;
   b1[25] := 0.0885571;
   b1[26] := 0.0390019;
   b1[27] := 0.075587;
   b1[28] := 0.1380671;
   b1[29] := 0.1447226;
   b1[30] := 0.048501;
   b1[31] := 0.1450995;
   w2[0] := 0.3448875;
   w2[1] := -0.0985299;
   w2[2] := -0.2385274;
   w2[3] := 0.1068773;
   w2[4] := 0.5171419;
   w2[5] := -0.1054032;
   w2[6] := 0.2936411;
   w2[7] := -0.4853331;
   w2[8] := -0.3005029;
   w2[9] := 0.2366145;
   w2[10] := 0.3783182;
   w2[11] := 0.127891;
   w2[12] := 0.0211917;
   w2[13] := -0.1069832;
   w2[14] := -0.2683547;
   w2[15] := -0.0976455;
   w2[16] := 0.6765909;
   w2[17] := 0.5036446;
   w2[18] := 0.3599868;
   w2[19] := 0.0810751;
   w2[20] := -0.079258;
   w2[21] := -0.2718676;
   w2[22] := -0.4316851;
   w2[23] := -0.1867653;
   w2[24] := 0.2037492;
   w2[25] := -0.0189868;
   w2[26] := -0.0119788;
   w2[27] := 0.3331117;
   w2[28] := -0.1736732;
   w2[29] := -0.4839838;
   w2[30] := -0.029798;
   w2[31] := -0.6352752;
   w2[32] := 0.4027197;
   w2[33] := -0.5263022;
   w2[34] := 0.2703936;
   w2[35] := 0.1180763;
   w2[36] := -0.3752257;
   w2[37] := -0.6156019;
   w2[38] := -0.4087748;
   w2[39] := 0.1517635;
   w2[40] := 0.2814839;
   w2[41] := -0.3188637;
   w2[42] := 0.4876765;
   w2[43] := 0.174788;
   w2[44] := -0.1799005;
   w2[45] := -0.3207765;
   w2[46] := 0.6545156;
   w2[47] := -0.3893254;
   w2[48] := -0.3369366;
   w2[49] := -0.437643;
   w2[50] := 0.041378;
   w2[51] := -0.1731163;
   w2[52] := 0.3791941;
   w2[53] := 0.0461393;
   w2[54] := 0.0816816;
   w2[55] := 0.3956819;
   w2[56] := -0.3843228;
   w2[57] := -0.7061806;
   w2[58] := -0.6190179;
   w2[59] := -0.4308152;
   w2[60] := 0.2132129;
   w2[61] := 0.4490756;
   w2[62] := -0.2397823;
   w2[63] := 0.3091693;
   w2[64] := -0.1736172;
   w2[65] := -0.6044765;
   w2[66] := 0.2081352;
   w2[67] := 0.4768652;
   w2[68] := -0.2759739;
   w2[69] := 0.1133698;
   w2[70] := -0.0100859;
   w2[71] := -0.6772556;
   w2[72] := 0.5169631;
   w2[73] := 0.1017481;
   w2[74] := -0.0672581;
   w2[75] := -0.4697476;
   w2[76] := -0.109866;
   w2[77] := -0.140197;
   w2[78] := -0.4618214;
   w2[79] := -0.2387714;
   w2[80] := -0.3492894;
   w2[81] := -0.2289385;
   w2[82] := 0.3859353;
   w2[83] := 0.3484918;
   w2[84] := 0.05708;
   w2[85] := 0.4838708;
   w2[86] := 0.441234;
   w2[87] := 0.1156965;
   w2[88] := 0.4213234;
   w2[89] := -0.2558614;
   w2[90] := 0.2997079;
   w2[91] := -0.0041088;
   w2[92] := -0.2610477;
   w2[93] := -0.2681805;
   w2[94] := 0.7025032;
   w2[95] := 0.403362;
   w2[96] := 0.0018223;
   w2[97] := 0.3965206;
   w2[98] := -0.113253;
   w2[99] := 0.3405365;
   w2[100] := 0.4333419;
   w2[101] := 0.0468351;
   w2[102] := -0.4313038;
   w2[103] := -0.5938676;
   w2[104] := -0.1057017;
   w2[105] := 0.3874305;
   w2[106] := -0.3047897;
   w2[107] := -0.360583;
   w2[108] := -0.0865778;
   w2[109] := 0.016962;
   w2[110] := -0.2818013;
   w2[111] := -0.205631;
   w2[112] := 0.2889744;
   w2[113] := -0.2389124;
   w2[114] := -0.5219849;
   w2[115] := -0.5379763;
   w2[116] := -0.3595321;
   w2[117] := 0.2131797;
   w2[118] := 0.2746126;
   w2[119] := 0.2555465;
   w2[120] := -0.3816569;
   w2[121] := -0.1742714;
   w2[122] := -0.3458711;
   w2[123] := -0.4732965;
   w2[124] := 0.3816739;
   w2[125] := 0.4522255;
   w2[126] := 0.4340182;
   w2[127] := 0.1317699;
   w2[128] := 0.0887004;
   w2[129] := -0.1704083;
   w2[130] := 0.2312619;
   w2[131] := -0.1512796;
   w2[132] := 0.1522121;
   w2[133] := -0.3580639;
   w2[134] := 0.3120518;
   w2[135] := -0.0891345;
   w2[136] := -0.5189782;
   w2[137] := 0.6759704;
   w2[138] := 0.8410841;
   w2[139] := -0.4388631;
   w2[140] := 0.3120123;
   w2[141] := 0.053066;
   w2[142] := -0.1540236;
   w2[143] := -0.1420563;
   w2[144] := 0.3882907;
   w2[145] := 0.3881267;
   w2[146] := 0.4476533;
   w2[147] := 0.4830106;
   w2[148] := 0.2335594;
   w2[149] := 0.1241002;
   w2[150] := -0.2032309;
   w2[151] := -0.5769788;
   w2[152] := 0.3601961;
   w2[153] := 0.5940281;
   w2[154] := -0.3626602;
   w2[155] := 0.1981693;
   w2[156] := -0.06857;
   w2[157] := -0.0704796;
   w2[158] := 0.0195035;
   w2[159] := -0.4674689;
   w2[160] := -0.2348353;
   w2[161] := -0.3250483;
   w2[162] := 0.1978887;
   w2[163] := -0.0533809;
   w2[164] := 0.5541837;
   w2[165] := 0.064756;
   w2[166] := 0.1574209;
   w2[167] := -0.4176951;
   w2[168] := -0.03289;
   w2[169] := -0.4697271;
   w2[170] := -0.0496295;
   w2[171] := -0.1912494;
   w2[172] := -0.2456453;
   w2[173] := -0.351849;
   w2[174] := 0.0067706;
   w2[175] := 0.6691334;
   w2[176] := 0.5995317;
   w2[177] := 0.3372136;
   w2[178] := -0.2781896;
   w2[179] := 0.2096184;
   w2[180] := -0.4983254;
   w2[181] := -0.0787928;
   w2[182] := -0.2063265;
   w2[183] := -0.2567849;
   w2[184] := -0.2985751;
   w2[185] := 0.2627156;
   w2[186] := 0.1459312;
   w2[187] := 0.4578165;
   w2[188] := 0.0136775;
   w2[189] := 0.4329558;
   w2[190] := -0.2819005;
   w2[191] := 0.077276;
   w2[192] := 0.1485205;
   w2[193] := 0.0424627;
   w2[194] := -0.5533946;
   w2[195] := -0.3114872;
   w2[196] := -0.0971009;
   w2[197] := 0.1043289;
   w2[198] := -0.0080725;
   w2[199] := 0.0561389;
   w2[200] := 0.1712011;
   w2[201] := -0.2093053;
   w2[202] := -0.4844932;
   w2[203] := 0.5200891;
   w2[204] := -0.4811763;
   w2[205] := -0.2097965;
   w2[206] := -0.1644997;
   w2[207] := 0.003576;
   w2[208] := 0.2773729;
   w2[209] := 0.4809147;
   w2[210] := -0.3132524;
   w2[211] := -0.0345517;
   w2[212] := 0.5111094;
   w2[213] := 0.1451371;
   w2[214] := 0.0575851;
   w2[215] := 0.1672285;
   w2[216] := 0.3724994;
   w2[217] := 0.0500904;
   w2[218] := -0.0895519;
   w2[219] := 0.0279228;
   w2[220] := -0.0756062;
   w2[221] := -0.6023685;
   w2[222] := 0.5966649;
   w2[223] := -0.4288191;
   w2[224] := -0.2491551;
   w2[225] := 0.1842164;
   w2[226] := 0.199599;
   w2[227] := 0.3348442;
   w2[228] := -0.6874152;
   w2[229] := 0.0923893;
   w2[230] := 0.5566139;
   w2[231] := 0.6076588;
   w2[232] := 0.4055642;
   w2[233] := 0.1035502;
   w2[234] := -0.2282035;
   w2[235] := 0.0315236;
   w2[236] := 0.3474;
   w2[237] := 0.1027276;
   w2[238] := 0.0550077;
   w2[239] := -0.1958367;
   w2[240] := -0.1637788;
   w2[241] := 0.2277053;
   w2[242] := -0.1716563;
   w2[243] := 0.1922517;
   w2[244] := 0.2188656;
   w2[245] := 0.0905953;
   w2[246] := -0.2237651;
   w2[247] := 0.4562837;
   w2[248] := -0.4297628;
   w2[249] := 0.0540233;
   w2[250] := -0.2155596;
   w2[251] := -0.4905677;
   w2[252] := 0.2578664;
   w2[253] := -0.0752592;
   w2[254] := 0.3203;
   w2[255] := 0.2922962;
   w2[256] := 0.6623323;
   w2[257] := -0.2237271;
   w2[258] := -0.378917;
   w2[259] := -0.3014932;
   w2[260] := 0.3499548;
   w2[261] := -0.3618023;
   w2[262] := -0.1381309;
   w2[263] := -0.2487616;
   w2[264] := -0.2042618;
   w2[265] := -0.3798007;
   w2[266] := 0.2168026;
   w2[267] := -0.5617495;
   w2[268] := 0.5470159;
   w2[269] := 0.3855161;
   w2[270] := -0.1744407;
   w2[271] := -0.0063227;
   w2[272] := -0.0175713;
   w2[273] := 0.4657946;
   w2[274] := 0.231147;
   w2[275] := 0.2995405;
   w2[276] := -0.2337339;
   w2[277] := 0.2714463;
   w2[278] := -0.1801859;
   w2[279] := -0.2387183;
   w2[280] := 0.2680195;
   w2[281] := 0.4208193;
   w2[282] := 0.0763752;
   w2[283] := -0.0259924;
   w2[284] := -0.5796329;
   w2[285] := -0.4459113;
   w2[286] := -0.0650182;
   w2[287] := 0.099238;
   w2[288] := -0.2287219;
   w2[289] := 0.1592736;
   w2[290] := 0.2655782;
   w2[291] := -0.7133095;
   w2[292] := -0.0750051;
   w2[293] := 0.1930008;
   w2[294] := 0.2515846;
   w2[295] := -0.104681;
   w2[296] := 0.3638516;
   w2[297] := -0.5185701;
   w2[298] := -0.137849;
   w2[299] := 0.1176404;
   w2[300] := -0.1728815;
   w2[301] := -0.4648141;
   w2[302] := -0.0106897;
   w2[303] := 0.2669196;
   w2[304] := -0.2057847;
   w2[305] := -0.0459625;
   w2[306] := -0.0872513;
   w2[307] := -0.5442434;
   w2[308] := 0.4806913;
   w2[309] := -0.2794292;
   w2[310] := 0.6181495;
   w2[311] := 0.4071167;
   w2[312] := -0.3071254;
   w2[313] := 0.1203253;
   w2[314] := 0.3505305;
   w2[315] := -0.5886531;
   w2[316] := -0.2951987;
   w2[317] := 0.3731146;
   w2[318] := 0.2878209;
   w2[319] := 0.24732;
   w2[320] := -0.1784255;
   w2[321] := 0.4152616;
   w2[322] := 0.505353;
   w2[323] := 0.2126275;
   w2[324] := 0.3228098;
   w2[325] := -0.3918779;
   w2[326] := -0.1658438;
   w2[327] := 0.5003296;
   w2[328] := -0.0053924;
   w2[329] := 0.0667791;
   w2[330] := 0.4097935;
   w2[331] := 0.1006095;
   w2[332] := 0.6046916;
   w2[333] := -0.0676274;
   w2[334] := -0.1915504;
   w2[335] := 0.3883604;
   w2[336] := 0.491134;
   w2[337] := 0.5468511;
   w2[338] := -0.1983627;
   w2[339] := -0.0676885;
   w2[340] := -0.3710055;
   w2[341] := 0.1606412;
   w2[342] := 0.4564988;
   w2[343] := -0.5501073;
   w2[344] := -0.1039538;
   w2[345] := -0.0296496;
   w2[346] := -0.5341417;
   w2[347] := -0.2000433;
   w2[348] := 0.2511403;
   w2[349] := 0.3043574;
   w2[350] := -0.1509714;
   w2[351] := 0.4652316;
   w2[352] := 0.5162573;
   w2[353] := -0.4559039;
   w2[354] := 0.155773;
   w2[355] := -0.3858083;
   w2[356] := 0.0727105;
   w2[357] := -0.4605626;
   w2[358] := -0.0643399;
   w2[359] := -0.2012528;
   w2[360] := -0.2376907;
   w2[361] := 0.633741;
   w2[362] := 0.7189264;
   w2[363] := 0.2091954;
   w2[364] := 0.7626936;
   w2[365] := 0.3527288;
   w2[366] := -0.1358239;
   w2[367] := 0.347225;
   w2[368] := -0.0854939;
   w2[369] := 0.3039412;
   w2[370] := 0.2409862;
   w2[371] := 0.4435183;
   w2[372] := 0.4328762;
   w2[373] := -0.02316;
   w2[374] := -0.117154;
   w2[375] := 0.0108573;
   w2[376] := -0.0911193;
   w2[377] := -0.5950353;
   w2[378] := -0.1391228;
   w2[379] := 0.1307337;
   w2[380] := -0.1149503;
   w2[381] := -0.0330209;
   w2[382] := -0.4081971;
   w2[383] := -0.3619282;
   w2[384] := -0.1067709;
   w2[385] := -0.0438268;
   w2[386] := 0.1861137;
   w2[387] := 0.1071503;
   w2[388] := -0.6722144;
   w2[389] := 0.5858943;
   w2[390] := 0.132711;
   w2[391] := 0.3459137;
   w2[392] := 0.3487434;
   w2[393] := 0.0373104;
   w2[394] := -0.256519;
   w2[395] := 0.4223759;
   w2[396] := -0.2403768;
   w2[397] := -0.0137525;
   w2[398] := 0.1307058;
   w2[399] := -0.5750338;
   w2[400] := -0.601782;
   w2[401] := 0.1216069;
   w2[402] := -0.0930582;
   w2[403] := 0.0528917;
   w2[404] := 0.2642088;
   w2[405] := 0.12135;
   w2[406] := -0.0773624;
   w2[407] := 0.1509228;
   w2[408] := 0.1637788;
   w2[409] := -0.0275139;
   w2[410] := 0.5865979;
   w2[411] := -0.2206961;
   w2[412] := 0.5099282;
   w2[413] := 0.2631257;
   w2[414] := 0.4237445;
   w2[415] := 0.4448525;
   w2[416] := 0.4446503;
   w2[417] := 0.0053865;
   w2[418] := -0.5579309;
   w2[419] := -0.1395655;
   w2[420] := -0.1579983;
   w2[421] := -0.3564516;
   w2[422] := 0.0891758;
   w2[423] := 0.1217025;
   w2[424] := -0.3250042;
   w2[425] := -0.0731721;
   w2[426] := 0.5731527;
   w2[427] := 0.3349074;
   w2[428] := -0.2764013;
   w2[429] := 0.3669565;
   w2[430] := 0.1658501;
   w2[431] := -0.0952915;
   w2[432] := 0.1848216;
   w2[433] := -0.3777516;
   w2[434] := 0.4125981;
   w2[435] := -0.2243889;
   w2[436] := 0.2011978;
   w2[437] := 0.3032005;
   w2[438] := 0.0724154;
   w2[439] := 0.2386405;
   w2[440] := -0.4659944;
   w2[441] := -0.5817581;
   w2[442] := -0.3680228;
   w2[443] := -0.5429725;
   w2[444] := -0.4282436;
   w2[445] := -0.0057439;
   w2[446] := 0.1407171;
   w2[447] := -0.0961595;
   w2[448] := -0.0304086;
   w2[449] := -0.559883;
   w2[450] := -0.5288109;
   w2[451] := 0.2501028;
   w2[452] := -0.1907448;
   w2[453] := 0.3364898;
   w2[454] := 0.3753116;
   w2[455] := -0.1153062;
   w2[456] := -0.0149126;
   w2[457] := -0.3870158;
   w2[458] := -0.115401;
   w2[459] := 0.0744122;
   w2[460] := -0.4487402;
   w2[461] := -0.2563244;
   w2[462] := 0.0335258;
   w2[463] := -0.1682583;
   w2[464] := 0.0443628;
   w2[465] := 0.3070406;
   w2[466] := -0.0503107;
   w2[467] := 0.0992935;
   w2[468] := 0.5251856;
   w2[469] := 0.6111719;
   w2[470] := 0.6419194;
   w2[471] := 0.1297791;
   w2[472] := 0.1860752;
   w2[473] := -0.1274762;
   w2[474] := 0.3434472;
   w2[475] := 0.550561;
   w2[476] := 0.3397494;
   w2[477] := -0.5685602;
   w2[478] := 0.0005795;
   w2[479] := -0.1080624;
   w2[480] := 0.3114881;
   w2[481] := 0.4475129;
   w2[482] := 0.1615055;
   w2[483] := -0.4390773;
   w2[484] := -0.0133804;
   w2[485] := -0.3265319;
   w2[486] := -0.598312;
   w2[487] := -0.2533576;
   w2[488] := 0.2004646;
   w2[489] := -0.2516977;
   w2[490] := -0.2211783;
   w2[491] := -0.0643062;
   w2[492] := 0.1233937;
   w2[493] := 0.1260124;
   w2[494] := -0.2689813;
   w2[495] := 0.3791626;
   w2[496] := 0.3063162;
   w2[497] := -0.2886556;
   w2[498] := -0.180589;
   w2[499] := -0.1727612;
   w2[500] := -0.2364416;
   w2[501] := -0.0335479;
   w2[502] := 0.1661869;
   w2[503] := 0.1447821;
   w2[504] := -0.1905543;
   w2[505] := -0.4342808;
   w2[506] := -0.0012427;
   w2[507] := -0.4948293;
   w2[508] := 0.0922625;
   w2[509] := 0.0781584;
   w2[510] := 0.4070034;
   w2[511] := 0.0575855;
   b3[0] := -0.0313972;
   b3[1] := -0.1867536;
   b3[2] := 0.2673712;
   b3[3] := 0.0710777;
   b3[4] := -0.2155338;
   b3[5] := 0.010384;
   b3[6] := 0.4061291;
   b3[7] := -0.0612305;
   b3[8] := 0.0899094;
   b3[9] := 0.1921517;
   b3[10] := 0.1069144;
   b3[11] := -0.0515455;
   b3[12] := 0.1089574;
   b3[13] := -0.1325741;
   b3[14] := 0.2726102;
   b3[15] := 0.1574048;
   w4[0] := -0.0865753;
   w4[1] := -0.5062438;
   w4[2] := 0.1554476;
   w4[3] := 0.7071172;
   w4[4] := -0.102356;
   w4[5] := 0.5811852;
   w4[6] := -0.6674285;
   w4[7] := -0.6164539;
   w4[8] := -0.810948;
   w4[9] := 0.6379222;
   w4[10] := 0.3449526;
   w4[11] := -0.0613255;
   w4[12] := -0.005266;
   w4[13] := -0.7050505;
   w4[14] := -0.6678494;
   w4[15] := 0.7979829;
   w4[16] := -0.0429653;
   w4[17] := -0.3721911;
   w4[18] := 0.9616893;
   w4[19] := -0.2787606;
   w4[20] := -0.1421925;
   w4[21] := -0.1321686;
   w4[22] := 0.1806948;
   w4[23] := -0.1417111;
   w4[24] := -0.4919258;
   w4[25] := 0.7062184;
   w4[26] := -0.488531;
   w4[27] := -0.5391713;
   w4[28] := 0.7159519;
   w4[29] := -0.5416421;
   w4[30] := 0.8190475;
   w4[31] := -0.2587632;
   w4[32] := 0.7209747;
   w4[33] := -0.5606546;
   w4[34] := 0.2996863;
   w4[35] := -0.4360698;
   w4[36] := 0.6557293;
   w4[37] := 0.7114502;
   w4[38] := -0.0711865;
   w4[39] := -0.5944882;
   w4[40] := 0.500967;
   w4[41] := -0.2733661;
   w4[42] := 0.0057439;
   w4[43] := 0.7727029;
   w4[44] := -0.5340657;
   w4[45] := 0.0551448;
   w4[46] := 0.2726173;
   w4[47] := -0.4893947;
   w4[48] := 0.286637;
   w4[49] := 0.6904863;
   w4[50] := -0.7133542;
   w4[51] := 0.1576146;
   w4[52] := 0.5721015;
   w4[53] := 0.0582882;
   w4[54] := -0.7719719;
   w4[55] := 0.2141585;
   w4[56] := -0.292623;
   w4[57] := -0.439004;
   w4[58] := 0.2077623;
   w4[59] := 0.5338089;
   w4[60] := 0.5839869;
   w4[61] := 0.7652564;
   w4[62] := -0.3743652;
   w4[63] := -0.1907377;
   b5[0] := -0.1430807;
   b5[1] := 0.2929625;
   b5[2] := 0.1342851;
   b5[3] := -0.1236853;
END_DATA_BLOCK

FUNCTION_BLOCK "TestFB"   // FB1, SCL
{ S7_Optimized_Access := 'FALSE' }
VERSION : 0.1
   VAR_INPUT
      idx : Int;
   END_VAR
   VAR_OUTPUT
      result : Real;
   END_VAR
BEGIN

       #result := "TestDB".test_arr[#idx];
END_FUNCTION_BLOCK

FUNCTION_BLOCK "NeuroPLC_Inference"   // FB2, SCL
{ S7_Optimized_Access := 'FALSE' }
VERSION : 0.1
// NeuroPLC 鈥?Auto-generated IEC 61131-3 SCL (DB+FB Mode)
//  Graph: mlp | Target: S71200DBBackend
//  Work memory: 75KB | LUT points: 0
//  Nodes: 8 | Ops: {'matmul': 4, 'standard_act': 2, 'softmax': 1, 'argmax': 1}
//  Parameters in DB "NeuroPLC_MLP_Weights", inference in FB.
   VAR_INPUT
      features : Array[0..27] of Real;   // 28-D feature vector
   END_VAR
   VAR_OUTPUT
      fault_class : Int;   // 0=Normal, 1=InnerRace, 2=Ball, 3=OuterRace
      confidence : Real;   // max softmax probability 鈹€鈹€ Inference temporaries 鈹€鈹€
   END_VAR
   VAR
      v1 : Array[0..31] of Real;   // matmul output
      v2 : Array[0..31] of Real;   // relu output
      v3 : Array[0..15] of Real;   // matmul output
      v4 : Array[0..15] of Real;   // relu output
      v5 : Array[0..3] of Real;   // matmul output
      v6 : Array[0..3] of Real;   // softmax output 鈹€鈹€ Temporary variables 鈹€鈹€
      i : Int;
      o : Int;
      j : Int;
      lo : Int;
      hi : Int;
      idx : Int;
      base : Int;
      sum : Real;
      max_val : Real;
      t_val : Real;
   END_VAR
BEGIN
      // 鈺愨晲鈺?Inference forward pass 鈺愨晲鈺?
       // Parameters loaded from DB "NeuroPLC_MLP_Weights" (start values = data, not code)

          // Input: features[0..27]

          // MatMul: fc0
          #v1[0] := "NeuroPLC_MLP_Weights".b1[0] + "NeuroPLC_MLP_Weights".w0[0] * #features[0] + "NeuroPLC_MLP_Weights".w0[1] * #features[1] + "NeuroPLC_MLP_Weights".w0[2] * #features[2] + "NeuroPLC_MLP_Weights".w0[3] * #features[3] + "NeuroPLC_MLP_Weights".w0[4] * #features[4] + "NeuroPLC_MLP_Weights".w0[5] * #features[5] + "NeuroPLC_MLP_Weights".w0[6] * #features[6] + "NeuroPLC_MLP_Weights".w0[7] * #features[7] + "NeuroPLC_MLP_Weights".w0[8] * #features[8] + "NeuroPLC_MLP_Weights".w0[9] * #features[9] + "NeuroPLC_MLP_Weights".w0[10] * #features[10] + "NeuroPLC_MLP_Weights".w0[11] * #features[11] + "NeuroPLC_MLP_Weights".w0[12] * #features[12] + "NeuroPLC_MLP_Weights".w0[13] * #features[13] + "NeuroPLC_MLP_Weights".w0[14] * #features[14] + "NeuroPLC_MLP_Weights".w0[15] * #features[15] + "NeuroPLC_MLP_Weights".w0[16] * #features[16] + "NeuroPLC_MLP_Weights".w0[17] * #features[17] + "NeuroPLC_MLP_Weights".w0[18] * #features[18] + "NeuroPLC_MLP_Weights".w0[19] * #features[19] + "NeuroPLC_MLP_Weights".w0[20] * #features[20] + "NeuroPLC_MLP_Weights".w0[21] * #features[21] + "NeuroPLC_MLP_Weights".w0[22] * #features[22] + "NeuroPLC_MLP_Weights".w0[23] * #features[23] + "NeuroPLC_MLP_Weights".w0[24] * #features[24] + "NeuroPLC_MLP_Weights".w0[25] * #features[25] + "NeuroPLC_MLP_Weights".w0[26] * #features[26] + "NeuroPLC_MLP_Weights".w0[27] * #features[27];
          #v1[1] := "NeuroPLC_MLP_Weights".b1[1] + "NeuroPLC_MLP_Weights".w0[28] * #features[0] + "NeuroPLC_MLP_Weights".w0[29] * #features[1] + "NeuroPLC_MLP_Weights".w0[30] * #features[2] + "NeuroPLC_MLP_Weights".w0[31] * #features[3] + "NeuroPLC_MLP_Weights".w0[32] * #features[4] + "NeuroPLC_MLP_Weights".w0[33] * #features[5] + "NeuroPLC_MLP_Weights".w0[34] * #features[6] + "NeuroPLC_MLP_Weights".w0[35] * #features[7] + "NeuroPLC_MLP_Weights".w0[36] * #features[8] + "NeuroPLC_MLP_Weights".w0[37] * #features[9] + "NeuroPLC_MLP_Weights".w0[38] * #features[10] + "NeuroPLC_MLP_Weights".w0[39] * #features[11] + "NeuroPLC_MLP_Weights".w0[40] * #features[12] + "NeuroPLC_MLP_Weights".w0[41] * #features[13] + "NeuroPLC_MLP_Weights".w0[42] * #features[14] + "NeuroPLC_MLP_Weights".w0[43] * #features[15] + "NeuroPLC_MLP_Weights".w0[44] * #features[16] + "NeuroPLC_MLP_Weights".w0[45] * #features[17] + "NeuroPLC_MLP_Weights".w0[46] * #features[18] + "NeuroPLC_MLP_Weights".w0[47] * #features[19] + "NeuroPLC_MLP_Weights".w0[48] * #features[20] + "NeuroPLC_MLP_Weights".w0[49] * #features[21] + "NeuroPLC_MLP_Weights".w0[50] * #features[22] + "NeuroPLC_MLP_Weights".w0[51] * #features[23] + "NeuroPLC_MLP_Weights".w0[52] * #features[24] + "NeuroPLC_MLP_Weights".w0[53] * #features[25] + "NeuroPLC_MLP_Weights".w0[54] * #features[26] + "NeuroPLC_MLP_Weights".w0[55] * #features[27];
          #v1[2] := "NeuroPLC_MLP_Weights".b1[2] + "NeuroPLC_MLP_Weights".w0[56] * #features[0] + "NeuroPLC_MLP_Weights".w0[57] * #features[1] + "NeuroPLC_MLP_Weights".w0[58] * #features[2] + "NeuroPLC_MLP_Weights".w0[59] * #features[3] + "NeuroPLC_MLP_Weights".w0[60] * #features[4] + "NeuroPLC_MLP_Weights".w0[61] * #features[5] + "NeuroPLC_MLP_Weights".w0[62] * #features[6] + "NeuroPLC_MLP_Weights".w0[63] * #features[7] + "NeuroPLC_MLP_Weights".w0[64] * #features[8] + "NeuroPLC_MLP_Weights".w0[65] * #features[9] + "NeuroPLC_MLP_Weights".w0[66] * #features[10] + "NeuroPLC_MLP_Weights".w0[67] * #features[11] + "NeuroPLC_MLP_Weights".w0[68] * #features[12] + "NeuroPLC_MLP_Weights".w0[69] * #features[13] + "NeuroPLC_MLP_Weights".w0[70] * #features[14] + "NeuroPLC_MLP_Weights".w0[71] * #features[15] + "NeuroPLC_MLP_Weights".w0[72] * #features[16] + "NeuroPLC_MLP_Weights".w0[73] * #features[17] + "NeuroPLC_MLP_Weights".w0[74] * #features[18] + "NeuroPLC_MLP_Weights".w0[75] * #features[19] + "NeuroPLC_MLP_Weights".w0[76] * #features[20] + "NeuroPLC_MLP_Weights".w0[77] * #features[21] + "NeuroPLC_MLP_Weights".w0[78] * #features[22] + "NeuroPLC_MLP_Weights".w0[79] * #features[23] + "NeuroPLC_MLP_Weights".w0[80] * #features[24] + "NeuroPLC_MLP_Weights".w0[81] * #features[25] + "NeuroPLC_MLP_Weights".w0[82] * #features[26] + "NeuroPLC_MLP_Weights".w0[83] * #features[27];
          #v1[3] := "NeuroPLC_MLP_Weights".b1[3] + "NeuroPLC_MLP_Weights".w0[84] * #features[0] + "NeuroPLC_MLP_Weights".w0[85] * #features[1] + "NeuroPLC_MLP_Weights".w0[86] * #features[2] + "NeuroPLC_MLP_Weights".w0[87] * #features[3] + "NeuroPLC_MLP_Weights".w0[88] * #features[4] + "NeuroPLC_MLP_Weights".w0[89] * #features[5] + "NeuroPLC_MLP_Weights".w0[90] * #features[6] + "NeuroPLC_MLP_Weights".w0[91] * #features[7] + "NeuroPLC_MLP_Weights".w0[92] * #features[8] + "NeuroPLC_MLP_Weights".w0[93] * #features[9] + "NeuroPLC_MLP_Weights".w0[94] * #features[10] + "NeuroPLC_MLP_Weights".w0[95] * #features[11] + "NeuroPLC_MLP_Weights".w0[96] * #features[12] + "NeuroPLC_MLP_Weights".w0[97] * #features[13] + "NeuroPLC_MLP_Weights".w0[98] * #features[14] + "NeuroPLC_MLP_Weights".w0[99] * #features[15] + "NeuroPLC_MLP_Weights".w0[100] * #features[16] + "NeuroPLC_MLP_Weights".w0[101] * #features[17] + "NeuroPLC_MLP_Weights".w0[102] * #features[18] + "NeuroPLC_MLP_Weights".w0[103] * #features[19] + "NeuroPLC_MLP_Weights".w0[104] * #features[20] + "NeuroPLC_MLP_Weights".w0[105] * #features[21] + "NeuroPLC_MLP_Weights".w0[106] * #features[22] + "NeuroPLC_MLP_Weights".w0[107] * #features[23] + "NeuroPLC_MLP_Weights".w0[108] * #features[24] + "NeuroPLC_MLP_Weights".w0[109] * #features[25] + "NeuroPLC_MLP_Weights".w0[110] * #features[26] + "NeuroPLC_MLP_Weights".w0[111] * #features[27];
          #v1[4] := "NeuroPLC_MLP_Weights".b1[4] + "NeuroPLC_MLP_Weights".w0[112] * #features[0] + "NeuroPLC_MLP_Weights".w0[113] * #features[1] + "NeuroPLC_MLP_Weights".w0[114] * #features[2] + "NeuroPLC_MLP_Weights".w0[115] * #features[3] + "NeuroPLC_MLP_Weights".w0[116] * #features[4] + "NeuroPLC_MLP_Weights".w0[117] * #features[5] + "NeuroPLC_MLP_Weights".w0[118] * #features[6] + "NeuroPLC_MLP_Weights".w0[119] * #features[7] + "NeuroPLC_MLP_Weights".w0[120] * #features[8] + "NeuroPLC_MLP_Weights".w0[121] * #features[9] + "NeuroPLC_MLP_Weights".w0[122] * #features[10] + "NeuroPLC_MLP_Weights".w0[123] * #features[11] + "NeuroPLC_MLP_Weights".w0[124] * #features[12] + "NeuroPLC_MLP_Weights".w0[125] * #features[13] + "NeuroPLC_MLP_Weights".w0[126] * #features[14] + "NeuroPLC_MLP_Weights".w0[127] * #features[15] + "NeuroPLC_MLP_Weights".w0[128] * #features[16] + "NeuroPLC_MLP_Weights".w0[129] * #features[17] + "NeuroPLC_MLP_Weights".w0[130] * #features[18] + "NeuroPLC_MLP_Weights".w0[131] * #features[19] + "NeuroPLC_MLP_Weights".w0[132] * #features[20] + "NeuroPLC_MLP_Weights".w0[133] * #features[21] + "NeuroPLC_MLP_Weights".w0[134] * #features[22] + "NeuroPLC_MLP_Weights".w0[135] * #features[23] + "NeuroPLC_MLP_Weights".w0[136] * #features[24] + "NeuroPLC_MLP_Weights".w0[137] * #features[25] + "NeuroPLC_MLP_Weights".w0[138] * #features[26] + "NeuroPLC_MLP_Weights".w0[139] * #features[27];
          #v1[5] := "NeuroPLC_MLP_Weights".b1[5] + "NeuroPLC_MLP_Weights".w0[140] * #features[0] + "NeuroPLC_MLP_Weights".w0[141] * #features[1] + "NeuroPLC_MLP_Weights".w0[142] * #features[2] + "NeuroPLC_MLP_Weights".w0[143] * #features[3] + "NeuroPLC_MLP_Weights".w0[144] * #features[4] + "NeuroPLC_MLP_Weights".w0[145] * #features[5] + "NeuroPLC_MLP_Weights".w0[146] * #features[6] + "NeuroPLC_MLP_Weights".w0[147] * #features[7] + "NeuroPLC_MLP_Weights".w0[148] * #features[8] + "NeuroPLC_MLP_Weights".w0[149] * #features[9] + "NeuroPLC_MLP_Weights".w0[150] * #features[10] + "NeuroPLC_MLP_Weights".w0[151] * #features[11] + "NeuroPLC_MLP_Weights".w0[152] * #features[12] + "NeuroPLC_MLP_Weights".w0[153] * #features[13] + "NeuroPLC_MLP_Weights".w0[154] * #features[14] + "NeuroPLC_MLP_Weights".w0[155] * #features[15] + "NeuroPLC_MLP_Weights".w0[156] * #features[16] + "NeuroPLC_MLP_Weights".w0[157] * #features[17] + "NeuroPLC_MLP_Weights".w0[158] * #features[18] + "NeuroPLC_MLP_Weights".w0[159] * #features[19] + "NeuroPLC_MLP_Weights".w0[160] * #features[20] + "NeuroPLC_MLP_Weights".w0[161] * #features[21] + "NeuroPLC_MLP_Weights".w0[162] * #features[22] + "NeuroPLC_MLP_Weights".w0[163] * #features[23] + "NeuroPLC_MLP_Weights".w0[164] * #features[24] + "NeuroPLC_MLP_Weights".w0[165] * #features[25] + "NeuroPLC_MLP_Weights".w0[166] * #features[26] + "NeuroPLC_MLP_Weights".w0[167] * #features[27];
          #v1[6] := "NeuroPLC_MLP_Weights".b1[6] + "NeuroPLC_MLP_Weights".w0[168] * #features[0] + "NeuroPLC_MLP_Weights".w0[169] * #features[1] + "NeuroPLC_MLP_Weights".w0[170] * #features[2] + "NeuroPLC_MLP_Weights".w0[171] * #features[3] + "NeuroPLC_MLP_Weights".w0[172] * #features[4] + "NeuroPLC_MLP_Weights".w0[173] * #features[5] + "NeuroPLC_MLP_Weights".w0[174] * #features[6] + "NeuroPLC_MLP_Weights".w0[175] * #features[7] + "NeuroPLC_MLP_Weights".w0[176] * #features[8] + "NeuroPLC_MLP_Weights".w0[177] * #features[9] + "NeuroPLC_MLP_Weights".w0[178] * #features[10] + "NeuroPLC_MLP_Weights".w0[179] * #features[11] + "NeuroPLC_MLP_Weights".w0[180] * #features[12] + "NeuroPLC_MLP_Weights".w0[181] * #features[13] + "NeuroPLC_MLP_Weights".w0[182] * #features[14] + "NeuroPLC_MLP_Weights".w0[183] * #features[15] + "NeuroPLC_MLP_Weights".w0[184] * #features[16] + "NeuroPLC_MLP_Weights".w0[185] * #features[17] + "NeuroPLC_MLP_Weights".w0[186] * #features[18] + "NeuroPLC_MLP_Weights".w0[187] * #features[19] + "NeuroPLC_MLP_Weights".w0[188] * #features[20] + "NeuroPLC_MLP_Weights".w0[189] * #features[21] + "NeuroPLC_MLP_Weights".w0[190] * #features[22] + "NeuroPLC_MLP_Weights".w0[191] * #features[23] + "NeuroPLC_MLP_Weights".w0[192] * #features[24] + "NeuroPLC_MLP_Weights".w0[193] * #features[25] + "NeuroPLC_MLP_Weights".w0[194] * #features[26] + "NeuroPLC_MLP_Weights".w0[195] * #features[27];
          #v1[7] := "NeuroPLC_MLP_Weights".b1[7] + "NeuroPLC_MLP_Weights".w0[196] * #features[0] + "NeuroPLC_MLP_Weights".w0[197] * #features[1] + "NeuroPLC_MLP_Weights".w0[198] * #features[2] + "NeuroPLC_MLP_Weights".w0[199] * #features[3] + "NeuroPLC_MLP_Weights".w0[200] * #features[4] + "NeuroPLC_MLP_Weights".w0[201] * #features[5] + "NeuroPLC_MLP_Weights".w0[202] * #features[6] + "NeuroPLC_MLP_Weights".w0[203] * #features[7] + "NeuroPLC_MLP_Weights".w0[204] * #features[8] + "NeuroPLC_MLP_Weights".w0[205] * #features[9] + "NeuroPLC_MLP_Weights".w0[206] * #features[10] + "NeuroPLC_MLP_Weights".w0[207] * #features[11] + "NeuroPLC_MLP_Weights".w0[208] * #features[12] + "NeuroPLC_MLP_Weights".w0[209] * #features[13] + "NeuroPLC_MLP_Weights".w0[210] * #features[14] + "NeuroPLC_MLP_Weights".w0[211] * #features[15] + "NeuroPLC_MLP_Weights".w0[212] * #features[16] + "NeuroPLC_MLP_Weights".w0[213] * #features[17] + "NeuroPLC_MLP_Weights".w0[214] * #features[18] + "NeuroPLC_MLP_Weights".w0[215] * #features[19] + "NeuroPLC_MLP_Weights".w0[216] * #features[20] + "NeuroPLC_MLP_Weights".w0[217] * #features[21] + "NeuroPLC_MLP_Weights".w0[218] * #features[22] + "NeuroPLC_MLP_Weights".w0[219] * #features[23] + "NeuroPLC_MLP_Weights".w0[220] * #features[24] + "NeuroPLC_MLP_Weights".w0[221] * #features[25] + "NeuroPLC_MLP_Weights".w0[222] * #features[26] + "NeuroPLC_MLP_Weights".w0[223] * #features[27];
          #v1[8] := "NeuroPLC_MLP_Weights".b1[8] + "NeuroPLC_MLP_Weights".w0[224] * #features[0] + "NeuroPLC_MLP_Weights".w0[225] * #features[1] + "NeuroPLC_MLP_Weights".w0[226] * #features[2] + "NeuroPLC_MLP_Weights".w0[227] * #features[3] + "NeuroPLC_MLP_Weights".w0[228] * #features[4] + "NeuroPLC_MLP_Weights".w0[229] * #features[5] + "NeuroPLC_MLP_Weights".w0[230] * #features[6] + "NeuroPLC_MLP_Weights".w0[231] * #features[7] + "NeuroPLC_MLP_Weights".w0[232] * #features[8] + "NeuroPLC_MLP_Weights".w0[233] * #features[9] + "NeuroPLC_MLP_Weights".w0[234] * #features[10] + "NeuroPLC_MLP_Weights".w0[235] * #features[11] + "NeuroPLC_MLP_Weights".w0[236] * #features[12] + "NeuroPLC_MLP_Weights".w0[237] * #features[13] + "NeuroPLC_MLP_Weights".w0[238] * #features[14] + "NeuroPLC_MLP_Weights".w0[239] * #features[15] + "NeuroPLC_MLP_Weights".w0[240] * #features[16] + "NeuroPLC_MLP_Weights".w0[241] * #features[17] + "NeuroPLC_MLP_Weights".w0[242] * #features[18] + "NeuroPLC_MLP_Weights".w0[243] * #features[19] + "NeuroPLC_MLP_Weights".w0[244] * #features[20] + "NeuroPLC_MLP_Weights".w0[245] * #features[21] + "NeuroPLC_MLP_Weights".w0[246] * #features[22] + "NeuroPLC_MLP_Weights".w0[247] * #features[23] + "NeuroPLC_MLP_Weights".w0[248] * #features[24] + "NeuroPLC_MLP_Weights".w0[249] * #features[25] + "NeuroPLC_MLP_Weights".w0[250] * #features[26] + "NeuroPLC_MLP_Weights".w0[251] * #features[27];
          #v1[9] := "NeuroPLC_MLP_Weights".b1[9] + "NeuroPLC_MLP_Weights".w0[252] * #features[0] + "NeuroPLC_MLP_Weights".w0[253] * #features[1] + "NeuroPLC_MLP_Weights".w0[254] * #features[2] + "NeuroPLC_MLP_Weights".w0[255] * #features[3] + "NeuroPLC_MLP_Weights".w0[256] * #features[4] + "NeuroPLC_MLP_Weights".w0[257] * #features[5] + "NeuroPLC_MLP_Weights".w0[258] * #features[6] + "NeuroPLC_MLP_Weights".w0[259] * #features[7] + "NeuroPLC_MLP_Weights".w0[260] * #features[8] + "NeuroPLC_MLP_Weights".w0[261] * #features[9] + "NeuroPLC_MLP_Weights".w0[262] * #features[10] + "NeuroPLC_MLP_Weights".w0[263] * #features[11] + "NeuroPLC_MLP_Weights".w0[264] * #features[12] + "NeuroPLC_MLP_Weights".w0[265] * #features[13] + "NeuroPLC_MLP_Weights".w0[266] * #features[14] + "NeuroPLC_MLP_Weights".w0[267] * #features[15] + "NeuroPLC_MLP_Weights".w0[268] * #features[16] + "NeuroPLC_MLP_Weights".w0[269] * #features[17] + "NeuroPLC_MLP_Weights".w0[270] * #features[18] + "NeuroPLC_MLP_Weights".w0[271] * #features[19] + "NeuroPLC_MLP_Weights".w0[272] * #features[20] + "NeuroPLC_MLP_Weights".w0[273] * #features[21] + "NeuroPLC_MLP_Weights".w0[274] * #features[22] + "NeuroPLC_MLP_Weights".w0[275] * #features[23] + "NeuroPLC_MLP_Weights".w0[276] * #features[24] + "NeuroPLC_MLP_Weights".w0[277] * #features[25] + "NeuroPLC_MLP_Weights".w0[278] * #features[26] + "NeuroPLC_MLP_Weights".w0[279] * #features[27];
          #v1[10] := "NeuroPLC_MLP_Weights".b1[10] + "NeuroPLC_MLP_Weights".w0[280] * #features[0] + "NeuroPLC_MLP_Weights".w0[281] * #features[1] + "NeuroPLC_MLP_Weights".w0[282] * #features[2] + "NeuroPLC_MLP_Weights".w0[283] * #features[3] + "NeuroPLC_MLP_Weights".w0[284] * #features[4] + "NeuroPLC_MLP_Weights".w0[285] * #features[5] + "NeuroPLC_MLP_Weights".w0[286] * #features[6] + "NeuroPLC_MLP_Weights".w0[287] * #features[7] + "NeuroPLC_MLP_Weights".w0[288] * #features[8] + "NeuroPLC_MLP_Weights".w0[289] * #features[9] + "NeuroPLC_MLP_Weights".w0[290] * #features[10] + "NeuroPLC_MLP_Weights".w0[291] * #features[11] + "NeuroPLC_MLP_Weights".w0[292] * #features[12] + "NeuroPLC_MLP_Weights".w0[293] * #features[13] + "NeuroPLC_MLP_Weights".w0[294] * #features[14] + "NeuroPLC_MLP_Weights".w0[295] * #features[15] + "NeuroPLC_MLP_Weights".w0[296] * #features[16] + "NeuroPLC_MLP_Weights".w0[297] * #features[17] + "NeuroPLC_MLP_Weights".w0[298] * #features[18] + "NeuroPLC_MLP_Weights".w0[299] * #features[19] + "NeuroPLC_MLP_Weights".w0[300] * #features[20] + "NeuroPLC_MLP_Weights".w0[301] * #features[21] + "NeuroPLC_MLP_Weights".w0[302] * #features[22] + "NeuroPLC_MLP_Weights".w0[303] * #features[23] + "NeuroPLC_MLP_Weights".w0[304] * #features[24] + "NeuroPLC_MLP_Weights".w0[305] * #features[25] + "NeuroPLC_MLP_Weights".w0[306] * #features[26] + "NeuroPLC_MLP_Weights".w0[307] * #features[27];
          #v1[11] := "NeuroPLC_MLP_Weights".b1[11] + "NeuroPLC_MLP_Weights".w0[308] * #features[0] + "NeuroPLC_MLP_Weights".w0[309] * #features[1] + "NeuroPLC_MLP_Weights".w0[310] * #features[2] + "NeuroPLC_MLP_Weights".w0[311] * #features[3] + "NeuroPLC_MLP_Weights".w0[312] * #features[4] + "NeuroPLC_MLP_Weights".w0[313] * #features[5] + "NeuroPLC_MLP_Weights".w0[314] * #features[6] + "NeuroPLC_MLP_Weights".w0[315] * #features[7] + "NeuroPLC_MLP_Weights".w0[316] * #features[8] + "NeuroPLC_MLP_Weights".w0[317] * #features[9] + "NeuroPLC_MLP_Weights".w0[318] * #features[10] + "NeuroPLC_MLP_Weights".w0[319] * #features[11] + "NeuroPLC_MLP_Weights".w0[320] * #features[12] + "NeuroPLC_MLP_Weights".w0[321] * #features[13] + "NeuroPLC_MLP_Weights".w0[322] * #features[14] + "NeuroPLC_MLP_Weights".w0[323] * #features[15] + "NeuroPLC_MLP_Weights".w0[324] * #features[16] + "NeuroPLC_MLP_Weights".w0[325] * #features[17] + "NeuroPLC_MLP_Weights".w0[326] * #features[18] + "NeuroPLC_MLP_Weights".w0[327] * #features[19] + "NeuroPLC_MLP_Weights".w0[328] * #features[20] + "NeuroPLC_MLP_Weights".w0[329] * #features[21] + "NeuroPLC_MLP_Weights".w0[330] * #features[22] + "NeuroPLC_MLP_Weights".w0[331] * #features[23] + "NeuroPLC_MLP_Weights".w0[332] * #features[24] + "NeuroPLC_MLP_Weights".w0[333] * #features[25] + "NeuroPLC_MLP_Weights".w0[334] * #features[26] + "NeuroPLC_MLP_Weights".w0[335] * #features[27];
          #v1[12] := "NeuroPLC_MLP_Weights".b1[12] + "NeuroPLC_MLP_Weights".w0[336] * #features[0] + "NeuroPLC_MLP_Weights".w0[337] * #features[1] + "NeuroPLC_MLP_Weights".w0[338] * #features[2] + "NeuroPLC_MLP_Weights".w0[339] * #features[3] + "NeuroPLC_MLP_Weights".w0[340] * #features[4] + "NeuroPLC_MLP_Weights".w0[341] * #features[5] + "NeuroPLC_MLP_Weights".w0[342] * #features[6] + "NeuroPLC_MLP_Weights".w0[343] * #features[7] + "NeuroPLC_MLP_Weights".w0[344] * #features[8] + "NeuroPLC_MLP_Weights".w0[345] * #features[9] + "NeuroPLC_MLP_Weights".w0[346] * #features[10] + "NeuroPLC_MLP_Weights".w0[347] * #features[11] + "NeuroPLC_MLP_Weights".w0[348] * #features[12] + "NeuroPLC_MLP_Weights".w0[349] * #features[13] + "NeuroPLC_MLP_Weights".w0[350] * #features[14] + "NeuroPLC_MLP_Weights".w0[351] * #features[15] + "NeuroPLC_MLP_Weights".w0[352] * #features[16] + "NeuroPLC_MLP_Weights".w0[353] * #features[17] + "NeuroPLC_MLP_Weights".w0[354] * #features[18] + "NeuroPLC_MLP_Weights".w0[355] * #features[19] + "NeuroPLC_MLP_Weights".w0[356] * #features[20] + "NeuroPLC_MLP_Weights".w0[357] * #features[21] + "NeuroPLC_MLP_Weights".w0[358] * #features[22] + "NeuroPLC_MLP_Weights".w0[359] * #features[23] + "NeuroPLC_MLP_Weights".w0[360] * #features[24] + "NeuroPLC_MLP_Weights".w0[361] * #features[25] + "NeuroPLC_MLP_Weights".w0[362] * #features[26] + "NeuroPLC_MLP_Weights".w0[363] * #features[27];
          #v1[13] := "NeuroPLC_MLP_Weights".b1[13] + "NeuroPLC_MLP_Weights".w0[364] * #features[0] + "NeuroPLC_MLP_Weights".w0[365] * #features[1] + "NeuroPLC_MLP_Weights".w0[366] * #features[2] + "NeuroPLC_MLP_Weights".w0[367] * #features[3] + "NeuroPLC_MLP_Weights".w0[368] * #features[4] + "NeuroPLC_MLP_Weights".w0[369] * #features[5] + "NeuroPLC_MLP_Weights".w0[370] * #features[6] + "NeuroPLC_MLP_Weights".w0[371] * #features[7] + "NeuroPLC_MLP_Weights".w0[372] * #features[8] + "NeuroPLC_MLP_Weights".w0[373] * #features[9] + "NeuroPLC_MLP_Weights".w0[374] * #features[10] + "NeuroPLC_MLP_Weights".w0[375] * #features[11] + "NeuroPLC_MLP_Weights".w0[376] * #features[12] + "NeuroPLC_MLP_Weights".w0[377] * #features[13] + "NeuroPLC_MLP_Weights".w0[378] * #features[14] + "NeuroPLC_MLP_Weights".w0[379] * #features[15] + "NeuroPLC_MLP_Weights".w0[380] * #features[16] + "NeuroPLC_MLP_Weights".w0[381] * #features[17] + "NeuroPLC_MLP_Weights".w0[382] * #features[18] + "NeuroPLC_MLP_Weights".w0[383] * #features[19] + "NeuroPLC_MLP_Weights".w0[384] * #features[20] + "NeuroPLC_MLP_Weights".w0[385] * #features[21] + "NeuroPLC_MLP_Weights".w0[386] * #features[22] + "NeuroPLC_MLP_Weights".w0[387] * #features[23] + "NeuroPLC_MLP_Weights".w0[388] * #features[24] + "NeuroPLC_MLP_Weights".w0[389] * #features[25] + "NeuroPLC_MLP_Weights".w0[390] * #features[26] + "NeuroPLC_MLP_Weights".w0[391] * #features[27];
          #v1[14] := "NeuroPLC_MLP_Weights".b1[14] + "NeuroPLC_MLP_Weights".w0[392] * #features[0] + "NeuroPLC_MLP_Weights".w0[393] * #features[1] + "NeuroPLC_MLP_Weights".w0[394] * #features[2] + "NeuroPLC_MLP_Weights".w0[395] * #features[3] + "NeuroPLC_MLP_Weights".w0[396] * #features[4] + "NeuroPLC_MLP_Weights".w0[397] * #features[5] + "NeuroPLC_MLP_Weights".w0[398] * #features[6] + "NeuroPLC_MLP_Weights".w0[399] * #features[7] + "NeuroPLC_MLP_Weights".w0[400] * #features[8] + "NeuroPLC_MLP_Weights".w0[401] * #features[9] + "NeuroPLC_MLP_Weights".w0[402] * #features[10] + "NeuroPLC_MLP_Weights".w0[403] * #features[11] + "NeuroPLC_MLP_Weights".w0[404] * #features[12] + "NeuroPLC_MLP_Weights".w0[405] * #features[13] + "NeuroPLC_MLP_Weights".w0[406] * #features[14] + "NeuroPLC_MLP_Weights".w0[407] * #features[15] + "NeuroPLC_MLP_Weights".w0[408] * #features[16] + "NeuroPLC_MLP_Weights".w0[409] * #features[17] + "NeuroPLC_MLP_Weights".w0[410] * #features[18] + "NeuroPLC_MLP_Weights".w0[411] * #features[19] + "NeuroPLC_MLP_Weights".w0[412] * #features[20] + "NeuroPLC_MLP_Weights".w0[413] * #features[21] + "NeuroPLC_MLP_Weights".w0[414] * #features[22] + "NeuroPLC_MLP_Weights".w0[415] * #features[23] + "NeuroPLC_MLP_Weights".w0[416] * #features[24] + "NeuroPLC_MLP_Weights".w0[417] * #features[25] + "NeuroPLC_MLP_Weights".w0[418] * #features[26] + "NeuroPLC_MLP_Weights".w0[419] * #features[27];
          #v1[15] := "NeuroPLC_MLP_Weights".b1[15] + "NeuroPLC_MLP_Weights".w0[420] * #features[0] + "NeuroPLC_MLP_Weights".w0[421] * #features[1] + "NeuroPLC_MLP_Weights".w0[422] * #features[2] + "NeuroPLC_MLP_Weights".w0[423] * #features[3] + "NeuroPLC_MLP_Weights".w0[424] * #features[4] + "NeuroPLC_MLP_Weights".w0[425] * #features[5] + "NeuroPLC_MLP_Weights".w0[426] * #features[6] + "NeuroPLC_MLP_Weights".w0[427] * #features[7] + "NeuroPLC_MLP_Weights".w0[428] * #features[8] + "NeuroPLC_MLP_Weights".w0[429] * #features[9] + "NeuroPLC_MLP_Weights".w0[430] * #features[10] + "NeuroPLC_MLP_Weights".w0[431] * #features[11] + "NeuroPLC_MLP_Weights".w0[432] * #features[12] + "NeuroPLC_MLP_Weights".w0[433] * #features[13] + "NeuroPLC_MLP_Weights".w0[434] * #features[14] + "NeuroPLC_MLP_Weights".w0[435] * #features[15] + "NeuroPLC_MLP_Weights".w0[436] * #features[16] + "NeuroPLC_MLP_Weights".w0[437] * #features[17] + "NeuroPLC_MLP_Weights".w0[438] * #features[18] + "NeuroPLC_MLP_Weights".w0[439] * #features[19] + "NeuroPLC_MLP_Weights".w0[440] * #features[20] + "NeuroPLC_MLP_Weights".w0[441] * #features[21] + "NeuroPLC_MLP_Weights".w0[442] * #features[22] + "NeuroPLC_MLP_Weights".w0[443] * #features[23] + "NeuroPLC_MLP_Weights".w0[444] * #features[24] + "NeuroPLC_MLP_Weights".w0[445] * #features[25] + "NeuroPLC_MLP_Weights".w0[446] * #features[26] + "NeuroPLC_MLP_Weights".w0[447] * #features[27];
          #v1[16] := "NeuroPLC_MLP_Weights".b1[16] + "NeuroPLC_MLP_Weights".w0[448] * #features[0] + "NeuroPLC_MLP_Weights".w0[449] * #features[1] + "NeuroPLC_MLP_Weights".w0[450] * #features[2] + "NeuroPLC_MLP_Weights".w0[451] * #features[3] + "NeuroPLC_MLP_Weights".w0[452] * #features[4] + "NeuroPLC_MLP_Weights".w0[453] * #features[5] + "NeuroPLC_MLP_Weights".w0[454] * #features[6] + "NeuroPLC_MLP_Weights".w0[455] * #features[7] + "NeuroPLC_MLP_Weights".w0[456] * #features[8] + "NeuroPLC_MLP_Weights".w0[457] * #features[9] + "NeuroPLC_MLP_Weights".w0[458] * #features[10] + "NeuroPLC_MLP_Weights".w0[459] * #features[11] + "NeuroPLC_MLP_Weights".w0[460] * #features[12] + "NeuroPLC_MLP_Weights".w0[461] * #features[13] + "NeuroPLC_MLP_Weights".w0[462] * #features[14] + "NeuroPLC_MLP_Weights".w0[463] * #features[15] + "NeuroPLC_MLP_Weights".w0[464] * #features[16] + "NeuroPLC_MLP_Weights".w0[465] * #features[17] + "NeuroPLC_MLP_Weights".w0[466] * #features[18] + "NeuroPLC_MLP_Weights".w0[467] * #features[19] + "NeuroPLC_MLP_Weights".w0[468] * #features[20] + "NeuroPLC_MLP_Weights".w0[469] * #features[21] + "NeuroPLC_MLP_Weights".w0[470] * #features[22] + "NeuroPLC_MLP_Weights".w0[471] * #features[23] + "NeuroPLC_MLP_Weights".w0[472] * #features[24] + "NeuroPLC_MLP_Weights".w0[473] * #features[25] + "NeuroPLC_MLP_Weights".w0[474] * #features[26] + "NeuroPLC_MLP_Weights".w0[475] * #features[27];
          #v1[17] := "NeuroPLC_MLP_Weights".b1[17] + "NeuroPLC_MLP_Weights".w0[476] * #features[0] + "NeuroPLC_MLP_Weights".w0[477] * #features[1] + "NeuroPLC_MLP_Weights".w0[478] * #features[2] + "NeuroPLC_MLP_Weights".w0[479] * #features[3] + "NeuroPLC_MLP_Weights".w0[480] * #features[4] + "NeuroPLC_MLP_Weights".w0[481] * #features[5] + "NeuroPLC_MLP_Weights".w0[482] * #features[6] + "NeuroPLC_MLP_Weights".w0[483] * #features[7] + "NeuroPLC_MLP_Weights".w0[484] * #features[8] + "NeuroPLC_MLP_Weights".w0[485] * #features[9] + "NeuroPLC_MLP_Weights".w0[486] * #features[10] + "NeuroPLC_MLP_Weights".w0[487] * #features[11] + "NeuroPLC_MLP_Weights".w0[488] * #features[12] + "NeuroPLC_MLP_Weights".w0[489] * #features[13] + "NeuroPLC_MLP_Weights".w0[490] * #features[14] + "NeuroPLC_MLP_Weights".w0[491] * #features[15] + "NeuroPLC_MLP_Weights".w0[492] * #features[16] + "NeuroPLC_MLP_Weights".w0[493] * #features[17] + "NeuroPLC_MLP_Weights".w0[494] * #features[18] + "NeuroPLC_MLP_Weights".w0[495] * #features[19] + "NeuroPLC_MLP_Weights".w0[496] * #features[20] + "NeuroPLC_MLP_Weights".w0[497] * #features[21] + "NeuroPLC_MLP_Weights".w0[498] * #features[22] + "NeuroPLC_MLP_Weights".w0[499] * #features[23] + "NeuroPLC_MLP_Weights".w0[500] * #features[24] + "NeuroPLC_MLP_Weights".w0[501] * #features[25] + "NeuroPLC_MLP_Weights".w0[502] * #features[26] + "NeuroPLC_MLP_Weights".w0[503] * #features[27];
          #v1[18] := "NeuroPLC_MLP_Weights".b1[18] + "NeuroPLC_MLP_Weights".w0[504] * #features[0] + "NeuroPLC_MLP_Weights".w0[505] * #features[1] + "NeuroPLC_MLP_Weights".w0[506] * #features[2] + "NeuroPLC_MLP_Weights".w0[507] * #features[3] + "NeuroPLC_MLP_Weights".w0[508] * #features[4] + "NeuroPLC_MLP_Weights".w0[509] * #features[5] + "NeuroPLC_MLP_Weights".w0[510] * #features[6] + "NeuroPLC_MLP_Weights".w0[511] * #features[7] + "NeuroPLC_MLP_Weights".w0[512] * #features[8] + "NeuroPLC_MLP_Weights".w0[513] * #features[9] + "NeuroPLC_MLP_Weights".w0[514] * #features[10] + "NeuroPLC_MLP_Weights".w0[515] * #features[11] + "NeuroPLC_MLP_Weights".w0[516] * #features[12] + "NeuroPLC_MLP_Weights".w0[517] * #features[13] + "NeuroPLC_MLP_Weights".w0[518] * #features[14] + "NeuroPLC_MLP_Weights".w0[519] * #features[15] + "NeuroPLC_MLP_Weights".w0[520] * #features[16] + "NeuroPLC_MLP_Weights".w0[521] * #features[17] + "NeuroPLC_MLP_Weights".w0[522] * #features[18] + "NeuroPLC_MLP_Weights".w0[523] * #features[19] + "NeuroPLC_MLP_Weights".w0[524] * #features[20] + "NeuroPLC_MLP_Weights".w0[525] * #features[21] + "NeuroPLC_MLP_Weights".w0[526] * #features[22] + "NeuroPLC_MLP_Weights".w0[527] * #features[23] + "NeuroPLC_MLP_Weights".w0[528] * #features[24] + "NeuroPLC_MLP_Weights".w0[529] * #features[25] + "NeuroPLC_MLP_Weights".w0[530] * #features[26] + "NeuroPLC_MLP_Weights".w0[531] * #features[27];
          #v1[19] := "NeuroPLC_MLP_Weights".b1[19] + "NeuroPLC_MLP_Weights".w0[532] * #features[0] + "NeuroPLC_MLP_Weights".w0[533] * #features[1] + "NeuroPLC_MLP_Weights".w0[534] * #features[2] + "NeuroPLC_MLP_Weights".w0[535] * #features[3] + "NeuroPLC_MLP_Weights".w0[536] * #features[4] + "NeuroPLC_MLP_Weights".w0[537] * #features[5] + "NeuroPLC_MLP_Weights".w0[538] * #features[6] + "NeuroPLC_MLP_Weights".w0[539] * #features[7] + "NeuroPLC_MLP_Weights".w0[540] * #features[8] + "NeuroPLC_MLP_Weights".w0[541] * #features[9] + "NeuroPLC_MLP_Weights".w0[542] * #features[10] + "NeuroPLC_MLP_Weights".w0[543] * #features[11] + "NeuroPLC_MLP_Weights".w0[544] * #features[12] + "NeuroPLC_MLP_Weights".w0[545] * #features[13] + "NeuroPLC_MLP_Weights".w0[546] * #features[14] + "NeuroPLC_MLP_Weights".w0[547] * #features[15] + "NeuroPLC_MLP_Weights".w0[548] * #features[16] + "NeuroPLC_MLP_Weights".w0[549] * #features[17] + "NeuroPLC_MLP_Weights".w0[550] * #features[18] + "NeuroPLC_MLP_Weights".w0[551] * #features[19] + "NeuroPLC_MLP_Weights".w0[552] * #features[20] + "NeuroPLC_MLP_Weights".w0[553] * #features[21] + "NeuroPLC_MLP_Weights".w0[554] * #features[22] + "NeuroPLC_MLP_Weights".w0[555] * #features[23] + "NeuroPLC_MLP_Weights".w0[556] * #features[24] + "NeuroPLC_MLP_Weights".w0[557] * #features[25] + "NeuroPLC_MLP_Weights".w0[558] * #features[26] + "NeuroPLC_MLP_Weights".w0[559] * #features[27];
          #v1[20] := "NeuroPLC_MLP_Weights".b1[20] + "NeuroPLC_MLP_Weights".w0[560] * #features[0] + "NeuroPLC_MLP_Weights".w0[561] * #features[1] + "NeuroPLC_MLP_Weights".w0[562] * #features[2] + "NeuroPLC_MLP_Weights".w0[563] * #features[3] + "NeuroPLC_MLP_Weights".w0[564] * #features[4] + "NeuroPLC_MLP_Weights".w0[565] * #features[5] + "NeuroPLC_MLP_Weights".w0[566] * #features[6] + "NeuroPLC_MLP_Weights".w0[567] * #features[7] + "NeuroPLC_MLP_Weights".w0[568] * #features[8] + "NeuroPLC_MLP_Weights".w0[569] * #features[9] + "NeuroPLC_MLP_Weights".w0[570] * #features[10] + "NeuroPLC_MLP_Weights".w0[571] * #features[11] + "NeuroPLC_MLP_Weights".w0[572] * #features[12] + "NeuroPLC_MLP_Weights".w0[573] * #features[13] + "NeuroPLC_MLP_Weights".w0[574] * #features[14] + "NeuroPLC_MLP_Weights".w0[575] * #features[15] + "NeuroPLC_MLP_Weights".w0[576] * #features[16] + "NeuroPLC_MLP_Weights".w0[577] * #features[17] + "NeuroPLC_MLP_Weights".w0[578] * #features[18] + "NeuroPLC_MLP_Weights".w0[579] * #features[19] + "NeuroPLC_MLP_Weights".w0[580] * #features[20] + "NeuroPLC_MLP_Weights".w0[581] * #features[21] + "NeuroPLC_MLP_Weights".w0[582] * #features[22] + "NeuroPLC_MLP_Weights".w0[583] * #features[23] + "NeuroPLC_MLP_Weights".w0[584] * #features[24] + "NeuroPLC_MLP_Weights".w0[585] * #features[25] + "NeuroPLC_MLP_Weights".w0[586] * #features[26] + "NeuroPLC_MLP_Weights".w0[587] * #features[27];
          #v1[21] := "NeuroPLC_MLP_Weights".b1[21] + "NeuroPLC_MLP_Weights".w0[588] * #features[0] + "NeuroPLC_MLP_Weights".w0[589] * #features[1] + "NeuroPLC_MLP_Weights".w0[590] * #features[2] + "NeuroPLC_MLP_Weights".w0[591] * #features[3] + "NeuroPLC_MLP_Weights".w0[592] * #features[4] + "NeuroPLC_MLP_Weights".w0[593] * #features[5] + "NeuroPLC_MLP_Weights".w0[594] * #features[6] + "NeuroPLC_MLP_Weights".w0[595] * #features[7] + "NeuroPLC_MLP_Weights".w0[596] * #features[8] + "NeuroPLC_MLP_Weights".w0[597] * #features[9] + "NeuroPLC_MLP_Weights".w0[598] * #features[10] + "NeuroPLC_MLP_Weights".w0[599] * #features[11] + "NeuroPLC_MLP_Weights".w0[600] * #features[12] + "NeuroPLC_MLP_Weights".w0[601] * #features[13] + "NeuroPLC_MLP_Weights".w0[602] * #features[14] + "NeuroPLC_MLP_Weights".w0[603] * #features[15] + "NeuroPLC_MLP_Weights".w0[604] * #features[16] + "NeuroPLC_MLP_Weights".w0[605] * #features[17] + "NeuroPLC_MLP_Weights".w0[606] * #features[18] + "NeuroPLC_MLP_Weights".w0[607] * #features[19] + "NeuroPLC_MLP_Weights".w0[608] * #features[20] + "NeuroPLC_MLP_Weights".w0[609] * #features[21] + "NeuroPLC_MLP_Weights".w0[610] * #features[22] + "NeuroPLC_MLP_Weights".w0[611] * #features[23] + "NeuroPLC_MLP_Weights".w0[612] * #features[24] + "NeuroPLC_MLP_Weights".w0[613] * #features[25] + "NeuroPLC_MLP_Weights".w0[614] * #features[26] + "NeuroPLC_MLP_Weights".w0[615] * #features[27];
          #v1[22] := "NeuroPLC_MLP_Weights".b1[22] + "NeuroPLC_MLP_Weights".w0[616] * #features[0] + "NeuroPLC_MLP_Weights".w0[617] * #features[1] + "NeuroPLC_MLP_Weights".w0[618] * #features[2] + "NeuroPLC_MLP_Weights".w0[619] * #features[3] + "NeuroPLC_MLP_Weights".w0[620] * #features[4] + "NeuroPLC_MLP_Weights".w0[621] * #features[5] + "NeuroPLC_MLP_Weights".w0[622] * #features[6] + "NeuroPLC_MLP_Weights".w0[623] * #features[7] + "NeuroPLC_MLP_Weights".w0[624] * #features[8] + "NeuroPLC_MLP_Weights".w0[625] * #features[9] + "NeuroPLC_MLP_Weights".w0[626] * #features[10] + "NeuroPLC_MLP_Weights".w0[627] * #features[11] + "NeuroPLC_MLP_Weights".w0[628] * #features[12] + "NeuroPLC_MLP_Weights".w0[629] * #features[13] + "NeuroPLC_MLP_Weights".w0[630] * #features[14] + "NeuroPLC_MLP_Weights".w0[631] * #features[15] + "NeuroPLC_MLP_Weights".w0[632] * #features[16] + "NeuroPLC_MLP_Weights".w0[633] * #features[17] + "NeuroPLC_MLP_Weights".w0[634] * #features[18] + "NeuroPLC_MLP_Weights".w0[635] * #features[19] + "NeuroPLC_MLP_Weights".w0[636] * #features[20] + "NeuroPLC_MLP_Weights".w0[637] * #features[21] + "NeuroPLC_MLP_Weights".w0[638] * #features[22] + "NeuroPLC_MLP_Weights".w0[639] * #features[23] + "NeuroPLC_MLP_Weights".w0[640] * #features[24] + "NeuroPLC_MLP_Weights".w0[641] * #features[25] + "NeuroPLC_MLP_Weights".w0[642] * #features[26] + "NeuroPLC_MLP_Weights".w0[643] * #features[27];
          #v1[23] := "NeuroPLC_MLP_Weights".b1[23] + "NeuroPLC_MLP_Weights".w0[644] * #features[0] + "NeuroPLC_MLP_Weights".w0[645] * #features[1] + "NeuroPLC_MLP_Weights".w0[646] * #features[2] + "NeuroPLC_MLP_Weights".w0[647] * #features[3] + "NeuroPLC_MLP_Weights".w0[648] * #features[4] + "NeuroPLC_MLP_Weights".w0[649] * #features[5] + "NeuroPLC_MLP_Weights".w0[650] * #features[6] + "NeuroPLC_MLP_Weights".w0[651] * #features[7] + "NeuroPLC_MLP_Weights".w0[652] * #features[8] + "NeuroPLC_MLP_Weights".w0[653] * #features[9] + "NeuroPLC_MLP_Weights".w0[654] * #features[10] + "NeuroPLC_MLP_Weights".w0[655] * #features[11] + "NeuroPLC_MLP_Weights".w0[656] * #features[12] + "NeuroPLC_MLP_Weights".w0[657] * #features[13] + "NeuroPLC_MLP_Weights".w0[658] * #features[14] + "NeuroPLC_MLP_Weights".w0[659] * #features[15] + "NeuroPLC_MLP_Weights".w0[660] * #features[16] + "NeuroPLC_MLP_Weights".w0[661] * #features[17] + "NeuroPLC_MLP_Weights".w0[662] * #features[18] + "NeuroPLC_MLP_Weights".w0[663] * #features[19] + "NeuroPLC_MLP_Weights".w0[664] * #features[20] + "NeuroPLC_MLP_Weights".w0[665] * #features[21] + "NeuroPLC_MLP_Weights".w0[666] * #features[22] + "NeuroPLC_MLP_Weights".w0[667] * #features[23] + "NeuroPLC_MLP_Weights".w0[668] * #features[24] + "NeuroPLC_MLP_Weights".w0[669] * #features[25] + "NeuroPLC_MLP_Weights".w0[670] * #features[26] + "NeuroPLC_MLP_Weights".w0[671] * #features[27];
          #v1[24] := "NeuroPLC_MLP_Weights".b1[24] + "NeuroPLC_MLP_Weights".w0[672] * #features[0] + "NeuroPLC_MLP_Weights".w0[673] * #features[1] + "NeuroPLC_MLP_Weights".w0[674] * #features[2] + "NeuroPLC_MLP_Weights".w0[675] * #features[3] + "NeuroPLC_MLP_Weights".w0[676] * #features[4] + "NeuroPLC_MLP_Weights".w0[677] * #features[5] + "NeuroPLC_MLP_Weights".w0[678] * #features[6] + "NeuroPLC_MLP_Weights".w0[679] * #features[7] + "NeuroPLC_MLP_Weights".w0[680] * #features[8] + "NeuroPLC_MLP_Weights".w0[681] * #features[9] + "NeuroPLC_MLP_Weights".w0[682] * #features[10] + "NeuroPLC_MLP_Weights".w0[683] * #features[11] + "NeuroPLC_MLP_Weights".w0[684] * #features[12] + "NeuroPLC_MLP_Weights".w0[685] * #features[13] + "NeuroPLC_MLP_Weights".w0[686] * #features[14] + "NeuroPLC_MLP_Weights".w0[687] * #features[15] + "NeuroPLC_MLP_Weights".w0[688] * #features[16] + "NeuroPLC_MLP_Weights".w0[689] * #features[17] + "NeuroPLC_MLP_Weights".w0[690] * #features[18] + "NeuroPLC_MLP_Weights".w0[691] * #features[19] + "NeuroPLC_MLP_Weights".w0[692] * #features[20] + "NeuroPLC_MLP_Weights".w0[693] * #features[21] + "NeuroPLC_MLP_Weights".w0[694] * #features[22] + "NeuroPLC_MLP_Weights".w0[695] * #features[23] + "NeuroPLC_MLP_Weights".w0[696] * #features[24] + "NeuroPLC_MLP_Weights".w0[697] * #features[25] + "NeuroPLC_MLP_Weights".w0[698] * #features[26] + "NeuroPLC_MLP_Weights".w0[699] * #features[27];
          #v1[25] := "NeuroPLC_MLP_Weights".b1[25] + "NeuroPLC_MLP_Weights".w0[700] * #features[0] + "NeuroPLC_MLP_Weights".w0[701] * #features[1] + "NeuroPLC_MLP_Weights".w0[702] * #features[2] + "NeuroPLC_MLP_Weights".w0[703] * #features[3] + "NeuroPLC_MLP_Weights".w0[704] * #features[4] + "NeuroPLC_MLP_Weights".w0[705] * #features[5] + "NeuroPLC_MLP_Weights".w0[706] * #features[6] + "NeuroPLC_MLP_Weights".w0[707] * #features[7] + "NeuroPLC_MLP_Weights".w0[708] * #features[8] + "NeuroPLC_MLP_Weights".w0[709] * #features[9] + "NeuroPLC_MLP_Weights".w0[710] * #features[10] + "NeuroPLC_MLP_Weights".w0[711] * #features[11] + "NeuroPLC_MLP_Weights".w0[712] * #features[12] + "NeuroPLC_MLP_Weights".w0[713] * #features[13] + "NeuroPLC_MLP_Weights".w0[714] * #features[14] + "NeuroPLC_MLP_Weights".w0[715] * #features[15] + "NeuroPLC_MLP_Weights".w0[716] * #features[16] + "NeuroPLC_MLP_Weights".w0[717] * #features[17] + "NeuroPLC_MLP_Weights".w0[718] * #features[18] + "NeuroPLC_MLP_Weights".w0[719] * #features[19] + "NeuroPLC_MLP_Weights".w0[720] * #features[20] + "NeuroPLC_MLP_Weights".w0[721] * #features[21] + "NeuroPLC_MLP_Weights".w0[722] * #features[22] + "NeuroPLC_MLP_Weights".w0[723] * #features[23] + "NeuroPLC_MLP_Weights".w0[724] * #features[24] + "NeuroPLC_MLP_Weights".w0[725] * #features[25] + "NeuroPLC_MLP_Weights".w0[726] * #features[26] + "NeuroPLC_MLP_Weights".w0[727] * #features[27];
          #v1[26] := "NeuroPLC_MLP_Weights".b1[26] + "NeuroPLC_MLP_Weights".w0[728] * #features[0] + "NeuroPLC_MLP_Weights".w0[729] * #features[1] + "NeuroPLC_MLP_Weights".w0[730] * #features[2] + "NeuroPLC_MLP_Weights".w0[731] * #features[3] + "NeuroPLC_MLP_Weights".w0[732] * #features[4] + "NeuroPLC_MLP_Weights".w0[733] * #features[5] + "NeuroPLC_MLP_Weights".w0[734] * #features[6] + "NeuroPLC_MLP_Weights".w0[735] * #features[7] + "NeuroPLC_MLP_Weights".w0[736] * #features[8] + "NeuroPLC_MLP_Weights".w0[737] * #features[9] + "NeuroPLC_MLP_Weights".w0[738] * #features[10] + "NeuroPLC_MLP_Weights".w0[739] * #features[11] + "NeuroPLC_MLP_Weights".w0[740] * #features[12] + "NeuroPLC_MLP_Weights".w0[741] * #features[13] + "NeuroPLC_MLP_Weights".w0[742] * #features[14] + "NeuroPLC_MLP_Weights".w0[743] * #features[15] + "NeuroPLC_MLP_Weights".w0[744] * #features[16] + "NeuroPLC_MLP_Weights".w0[745] * #features[17] + "NeuroPLC_MLP_Weights".w0[746] * #features[18] + "NeuroPLC_MLP_Weights".w0[747] * #features[19] + "NeuroPLC_MLP_Weights".w0[748] * #features[20] + "NeuroPLC_MLP_Weights".w0[749] * #features[21] + "NeuroPLC_MLP_Weights".w0[750] * #features[22] + "NeuroPLC_MLP_Weights".w0[751] * #features[23] + "NeuroPLC_MLP_Weights".w0[752] * #features[24] + "NeuroPLC_MLP_Weights".w0[753] * #features[25] + "NeuroPLC_MLP_Weights".w0[754] * #features[26] + "NeuroPLC_MLP_Weights".w0[755] * #features[27];
          #v1[27] := "NeuroPLC_MLP_Weights".b1[27] + "NeuroPLC_MLP_Weights".w0[756] * #features[0] + "NeuroPLC_MLP_Weights".w0[757] * #features[1] + "NeuroPLC_MLP_Weights".w0[758] * #features[2] + "NeuroPLC_MLP_Weights".w0[759] * #features[3] + "NeuroPLC_MLP_Weights".w0[760] * #features[4] + "NeuroPLC_MLP_Weights".w0[761] * #features[5] + "NeuroPLC_MLP_Weights".w0[762] * #features[6] + "NeuroPLC_MLP_Weights".w0[763] * #features[7] + "NeuroPLC_MLP_Weights".w0[764] * #features[8] + "NeuroPLC_MLP_Weights".w0[765] * #features[9] + "NeuroPLC_MLP_Weights".w0[766] * #features[10] + "NeuroPLC_MLP_Weights".w0[767] * #features[11] + "NeuroPLC_MLP_Weights".w0[768] * #features[12] + "NeuroPLC_MLP_Weights".w0[769] * #features[13] + "NeuroPLC_MLP_Weights".w0[770] * #features[14] + "NeuroPLC_MLP_Weights".w0[771] * #features[15] + "NeuroPLC_MLP_Weights".w0[772] * #features[16] + "NeuroPLC_MLP_Weights".w0[773] * #features[17] + "NeuroPLC_MLP_Weights".w0[774] * #features[18] + "NeuroPLC_MLP_Weights".w0[775] * #features[19] + "NeuroPLC_MLP_Weights".w0[776] * #features[20] + "NeuroPLC_MLP_Weights".w0[777] * #features[21] + "NeuroPLC_MLP_Weights".w0[778] * #features[22] + "NeuroPLC_MLP_Weights".w0[779] * #features[23] + "NeuroPLC_MLP_Weights".w0[780] * #features[24] + "NeuroPLC_MLP_Weights".w0[781] * #features[25] + "NeuroPLC_MLP_Weights".w0[782] * #features[26] + "NeuroPLC_MLP_Weights".w0[783] * #features[27];
          #v1[28] := "NeuroPLC_MLP_Weights".b1[28] + "NeuroPLC_MLP_Weights".w0[784] * #features[0] + "NeuroPLC_MLP_Weights".w0[785] * #features[1] + "NeuroPLC_MLP_Weights".w0[786] * #features[2] + "NeuroPLC_MLP_Weights".w0[787] * #features[3] + "NeuroPLC_MLP_Weights".w0[788] * #features[4] + "NeuroPLC_MLP_Weights".w0[789] * #features[5] + "NeuroPLC_MLP_Weights".w0[790] * #features[6] + "NeuroPLC_MLP_Weights".w0[791] * #features[7] + "NeuroPLC_MLP_Weights".w0[792] * #features[8] + "NeuroPLC_MLP_Weights".w0[793] * #features[9] + "NeuroPLC_MLP_Weights".w0[794] * #features[10] + "NeuroPLC_MLP_Weights".w0[795] * #features[11] + "NeuroPLC_MLP_Weights".w0[796] * #features[12] + "NeuroPLC_MLP_Weights".w0[797] * #features[13] + "NeuroPLC_MLP_Weights".w0[798] * #features[14] + "NeuroPLC_MLP_Weights".w0[799] * #features[15] + "NeuroPLC_MLP_Weights".w0[800] * #features[16] + "NeuroPLC_MLP_Weights".w0[801] * #features[17] + "NeuroPLC_MLP_Weights".w0[802] * #features[18] + "NeuroPLC_MLP_Weights".w0[803] * #features[19] + "NeuroPLC_MLP_Weights".w0[804] * #features[20] + "NeuroPLC_MLP_Weights".w0[805] * #features[21] + "NeuroPLC_MLP_Weights".w0[806] * #features[22] + "NeuroPLC_MLP_Weights".w0[807] * #features[23] + "NeuroPLC_MLP_Weights".w0[808] * #features[24] + "NeuroPLC_MLP_Weights".w0[809] * #features[25] + "NeuroPLC_MLP_Weights".w0[810] * #features[26] + "NeuroPLC_MLP_Weights".w0[811] * #features[27];
          #v1[29] := "NeuroPLC_MLP_Weights".b1[29] + "NeuroPLC_MLP_Weights".w0[812] * #features[0] + "NeuroPLC_MLP_Weights".w0[813] * #features[1] + "NeuroPLC_MLP_Weights".w0[814] * #features[2] + "NeuroPLC_MLP_Weights".w0[815] * #features[3] + "NeuroPLC_MLP_Weights".w0[816] * #features[4] + "NeuroPLC_MLP_Weights".w0[817] * #features[5] + "NeuroPLC_MLP_Weights".w0[818] * #features[6] + "NeuroPLC_MLP_Weights".w0[819] * #features[7] + "NeuroPLC_MLP_Weights".w0[820] * #features[8] + "NeuroPLC_MLP_Weights".w0[821] * #features[9] + "NeuroPLC_MLP_Weights".w0[822] * #features[10] + "NeuroPLC_MLP_Weights".w0[823] * #features[11] + "NeuroPLC_MLP_Weights".w0[824] * #features[12] + "NeuroPLC_MLP_Weights".w0[825] * #features[13] + "NeuroPLC_MLP_Weights".w0[826] * #features[14] + "NeuroPLC_MLP_Weights".w0[827] * #features[15] + "NeuroPLC_MLP_Weights".w0[828] * #features[16] + "NeuroPLC_MLP_Weights".w0[829] * #features[17] + "NeuroPLC_MLP_Weights".w0[830] * #features[18] + "NeuroPLC_MLP_Weights".w0[831] * #features[19] + "NeuroPLC_MLP_Weights".w0[832] * #features[20] + "NeuroPLC_MLP_Weights".w0[833] * #features[21] + "NeuroPLC_MLP_Weights".w0[834] * #features[22] + "NeuroPLC_MLP_Weights".w0[835] * #features[23] + "NeuroPLC_MLP_Weights".w0[836] * #features[24] + "NeuroPLC_MLP_Weights".w0[837] * #features[25] + "NeuroPLC_MLP_Weights".w0[838] * #features[26] + "NeuroPLC_MLP_Weights".w0[839] * #features[27];
          #v1[30] := "NeuroPLC_MLP_Weights".b1[30] + "NeuroPLC_MLP_Weights".w0[840] * #features[0] + "NeuroPLC_MLP_Weights".w0[841] * #features[1] + "NeuroPLC_MLP_Weights".w0[842] * #features[2] + "NeuroPLC_MLP_Weights".w0[843] * #features[3] + "NeuroPLC_MLP_Weights".w0[844] * #features[4] + "NeuroPLC_MLP_Weights".w0[845] * #features[5] + "NeuroPLC_MLP_Weights".w0[846] * #features[6] + "NeuroPLC_MLP_Weights".w0[847] * #features[7] + "NeuroPLC_MLP_Weights".w0[848] * #features[8] + "NeuroPLC_MLP_Weights".w0[849] * #features[9] + "NeuroPLC_MLP_Weights".w0[850] * #features[10] + "NeuroPLC_MLP_Weights".w0[851] * #features[11] + "NeuroPLC_MLP_Weights".w0[852] * #features[12] + "NeuroPLC_MLP_Weights".w0[853] * #features[13] + "NeuroPLC_MLP_Weights".w0[854] * #features[14] + "NeuroPLC_MLP_Weights".w0[855] * #features[15] + "NeuroPLC_MLP_Weights".w0[856] * #features[16] + "NeuroPLC_MLP_Weights".w0[857] * #features[17] + "NeuroPLC_MLP_Weights".w0[858] * #features[18] + "NeuroPLC_MLP_Weights".w0[859] * #features[19] + "NeuroPLC_MLP_Weights".w0[860] * #features[20] + "NeuroPLC_MLP_Weights".w0[861] * #features[21] + "NeuroPLC_MLP_Weights".w0[862] * #features[22] + "NeuroPLC_MLP_Weights".w0[863] * #features[23] + "NeuroPLC_MLP_Weights".w0[864] * #features[24] + "NeuroPLC_MLP_Weights".w0[865] * #features[25] + "NeuroPLC_MLP_Weights".w0[866] * #features[26] + "NeuroPLC_MLP_Weights".w0[867] * #features[27];
          #v1[31] := "NeuroPLC_MLP_Weights".b1[31] + "NeuroPLC_MLP_Weights".w0[868] * #features[0] + "NeuroPLC_MLP_Weights".w0[869] * #features[1] + "NeuroPLC_MLP_Weights".w0[870] * #features[2] + "NeuroPLC_MLP_Weights".w0[871] * #features[3] + "NeuroPLC_MLP_Weights".w0[872] * #features[4] + "NeuroPLC_MLP_Weights".w0[873] * #features[5] + "NeuroPLC_MLP_Weights".w0[874] * #features[6] + "NeuroPLC_MLP_Weights".w0[875] * #features[7] + "NeuroPLC_MLP_Weights".w0[876] * #features[8] + "NeuroPLC_MLP_Weights".w0[877] * #features[9] + "NeuroPLC_MLP_Weights".w0[878] * #features[10] + "NeuroPLC_MLP_Weights".w0[879] * #features[11] + "NeuroPLC_MLP_Weights".w0[880] * #features[12] + "NeuroPLC_MLP_Weights".w0[881] * #features[13] + "NeuroPLC_MLP_Weights".w0[882] * #features[14] + "NeuroPLC_MLP_Weights".w0[883] * #features[15] + "NeuroPLC_MLP_Weights".w0[884] * #features[16] + "NeuroPLC_MLP_Weights".w0[885] * #features[17] + "NeuroPLC_MLP_Weights".w0[886] * #features[18] + "NeuroPLC_MLP_Weights".w0[887] * #features[19] + "NeuroPLC_MLP_Weights".w0[888] * #features[20] + "NeuroPLC_MLP_Weights".w0[889] * #features[21] + "NeuroPLC_MLP_Weights".w0[890] * #features[22] + "NeuroPLC_MLP_Weights".w0[891] * #features[23] + "NeuroPLC_MLP_Weights".w0[892] * #features[24] + "NeuroPLC_MLP_Weights".w0[893] * #features[25] + "NeuroPLC_MLP_Weights".w0[894] * #features[26] + "NeuroPLC_MLP_Weights".w0[895] * #features[27];

          // StandardAct: relu
          FOR #i := 0 TO 31 DO
              IF #v1[#i] < 0.0 THEN
                  #v2[#i] := 0.0;
              ELSE
                  #v2[#i] := #v1[#i];
              END_IF;
          END_FOR;

